Fanuc TP program (LS listing): OP5_LRG_MASTER_AIR_F.LS

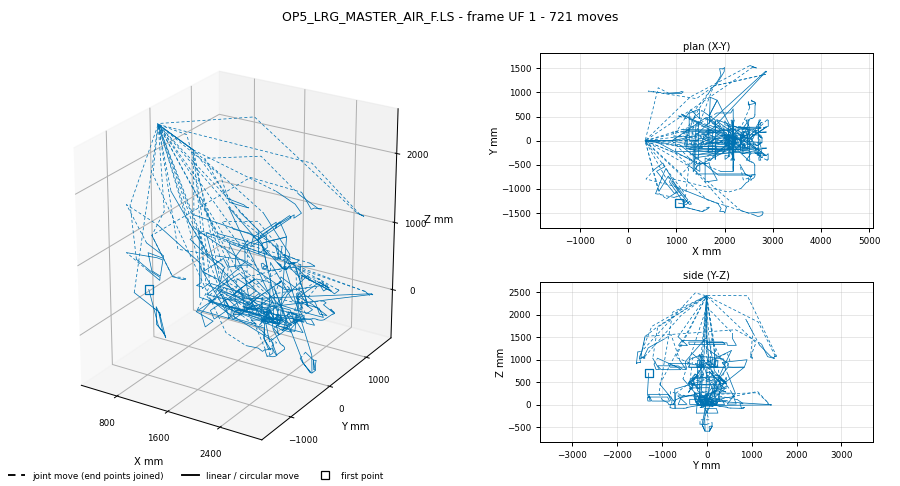
[picture p0: tool path of OP5_LRG_MASTER_AIR_F.LS in frame UF 1, 721 of 721 moves have a stored position in this frame; points joined in program order, loops and branches not executed]
/PROG  OP5_LRG_MASTER_AIR_F
/ATTR
OWNER		= MNEDITOR;
COMMENT		= "Air move update";
PROG_SIZE	= 123886;
CREATE		= DATE 25-08-25  TIME 10:39:22;
MODIFIED	= DATE 25-08-25  TIME 10:43:36;
FILE_NAME	= OP5_LRG_;
VERSION		= 0;
LINE_COUNT	= 2640;
MEMORY_SIZE	= 124514;
PROTECT		= READ_WRITE;
TCD:  STACK_SIZE	= 0,
      TASK_PRIORITY	= 50,
      TIME_SLICE	= 0,
      BUSY_LAMP_OFF	= 0,
      ABORT_REQUEST	= 0,
      PAUSE_REQUEST	= 0;
DEFAULT_GROUP	= 1,1,*,*,*;
CONTROL_CODE	= 00000000 00000000;
/APPL
  ARC Welding Equipment : 1,*,*,*,*;

MPAS ;
MPAS_NUM_PASSES        : 0;
MPAS_LAST_PASS         : 0;
MPAS_CURRENT_PASS      : 0;
MPAS_STATUS_PASS       : 0;
/MN
   1:  !********** WAR HAMMER ********** ;
   2:  !*------- FRAME LARGE ----------* ;
   3:  !*------- FR500 CELL: F --------* ;
   4:  !******************************** ;
   5:   ;
   6:  CALL HOME    ;
   7:  UFRAME_NUM=1 ;
   8:  DO[17:ON :SCAN ZONE2]=OFF ;
   9:   ;
  10:  !********POSITIONER MOVE******** ;
  11:J P[1] 85% CNT30    ;
  12:   ;
  13:L P[3] 1000mm/sec CNT40    ;
  14:   ;
  15:  !FR50L1000 ;
  16:  IF R[15:TECH HOLD]=1002,CALL TECH_HOLD ;
  17:   ;
  18:  !TO SKIP FRONT BUMPER WELDS ;
  19:  CALL ARC_DISABLE_FRONT_BMPR_LRG(0) ;
  20:   ;
1578:   ;
1579:L P[124] 1000mm/sec FINE
    :  Arc Start[6]    ;
1580:  Weave Sine[6] ;
1581:  Track TAST[6] ;
1582:L P[125] WELD_SPEED FINE
    :  Arc End[6]    ;
1583:  Weave End ;
1584:  Track End ;
1585:   ;
  22:   ;
  23:   ;
  24:L P[8] 800mm/sec CNT30    ;
  25:   ;
  26:L P[9] 1000mm/sec CNT30    ;
  27:   ;
  28:   ;
  29:  !FR50L1001 ;
  30:  IF R[15:TECH HOLD]=1003,CALL TECH_HOLD ;
  31:   ;
  32:   ;
1587:   ;
1588:L P[126] 1000mm/sec FINE
    :  Arc Start[6]    ;
1589:  Weave Sine[6] ;
1590:  Track TAST[6] ;
1591:L P[129] WELD_SPEED FINE
    :  Arc End[6]    ;
1592:  Weave End ;
1593:  Track End ;
1594:   ;
  34:   ;
  35:L P[12] 1000mm/sec CNT100    ;
  36:   ;
  37:   ;
  38:  !FR50L1002 ;
  39:  IF R[15:TECH HOLD]=1004,CALL TECH_HOLD ;
  40:   ;
  41:   ;
  42:L P[13] 1000mm/sec CNT70    ;
  43:   ;
1596:   ;
1597:L P[130] 1000mm/sec FINE
    :  Arc Start[6]    ;
1598:  Weave Sine[6] ;
1599:  Track TAST[6] ;
1600:L P[131] WELD_SPEED FINE
    :  Arc End[6]    ;
1601:  Weave End ;
1602:  Track End ;
1603:   ;
  45:   ;
  46:  CALL ARC_DISABLE_FRONT_BMPR_LRG(1) ;
  47:   ;
  48:L P[16] 1000mm/sec CNT100    ;
  49:   ;
  50:  !HOME ;
  51:J P[4] 70% CNT30    ;
  52:   ;
  53:  !********POSITIONER MOVE******** ;
  54:J P[17] 85% CNT30    ;
  55:   ;
  56:J P[18] 50% CNT100    ;
  57:   ;
  58:L P[19] 1000mm/sec CNT100    ;
  59:   ;
  60:   ;
  61:  !FR50L1003 ;
  62:  IF R[15:TECH HOLD]=1005,CALL TECH_HOLD ;
  63:   ;
  64:   ;
  65:L P[20] 1000mm/sec CNT25    ;
  66:   ;
1605:   ;
1606:L P[132] 1000mm/sec FINE
    :  Arc Start[6]    ;
1607:  Weave Sine[6] ;
1608:  Track TAST[6] ;
1609:L P[137] WELD_SPEED CNT100    ;
1610:L P[138] WELD_SPEED FINE
    :  Arc End[6]    ;
1611:  Track End ;
1612:  Weave End ;
1613:   ;
  68:   ;
  69:L P[24] 1000mm/sec CNT30    ;
  70:   ;
  71:   ;
  72:  !FR50L1010 ;
  73:  IF R[15:TECH HOLD]=1012,CALL TECH_HOLD ;
  74:   ;
  75:   ;
  76:L P[25] 1000mm/sec CNT30    ;
  77:   ;
1615:   ;
1616:L P[141] 1000mm/sec FINE
    :  Arc Start[6]    ;
1617:  Weave Sine[6] ;
1618:  Track TAST[6] ;
1619:L P[142] WELD_SPEED CNT100    ;
1620:L P[146] WELD_SPEED FINE
    :  Arc End[6]    ;
1621:  Weave End ;
1622:  Track End ;
1623:   ;
  79:   ;
  80:L P[29] 1000mm/sec CNT25    ;
  81:   ;
  82:   ;
  83:  !FR50L1020 ;
  84:  IF R[15:TECH HOLD]=1022,CALL TECH_HOLD ;
  85:   ;
  86:   ;
  87:J P[30] 50% CNT25    ;
  88:   ;
1625:   ;
1626:L P[147] 1000mm/sec FINE
    :  Arc Start[6]    ;
1627:  Weave Sine[6] ;
1628:  Track TAST[6] ;
1629:L P[150] WELD_SPEED FINE
    :  Arc End[6]    ;
1630:  Weave End ;
1631:  Track End ;
1632:   ;
  90:   ;
  91:L P[33] 1000mm/sec CNT30    ;
  92:   ;
  93:L P[34] 1000mm/sec CNT30    ;
  94:   ;
  95:   ;
  96:  !FR50L1030 ;
  97:  IF R[15:TECH HOLD]=1032,CALL TECH_HOLD ;
  98:   ;
  99:   ;
1634:   ;
1635:L P[151] 1000mm/sec FINE
    :  Arc Start[6]    ;
1636:  Weave Sine[6] ;
1637:  Track TAST[6] ;
1638:L P[156] WELD_SPEED FINE
    :  Arc End[6]    ;
1639:  Weave End ;
1640:  Track End ;
1641:   ;
 101:   ;
 102:L P[37] 1000mm/sec CNT50    ;
 103:   ;
 104:J P[38] 50% CNT50    ;
 105:   ;
 106:L P[39] 1000mm/sec CNT25    ;
 107:   ;
 108:   ;
 109:  !FR50L1040 ;
 110:  IF R[15:TECH HOLD]=1042,CALL TECH_HOLD ;
 111:   ;
 112:   ;
1643:   ;
1644:L P[157] 1000mm/sec FINE
    :  Arc Start[6]    ;
1645:  Weave Sine[6] ;
1646:L P[158] WELD_SPEED FINE
    :  Arc End[6]    ;
1647:  Weave End ;
1648:   ;
 114:   ;
 115:L P[42] 1000mm/sec CNT30    ;
 116:   ;
 117:L P[43] 1000mm/sec CNT70    ;
 118:   ;
 119:J P[44] 50% CNT50    ;
 120:   ;
 121:L P[45] 1000mm/sec CNT30    ;
 122:   ;
 123:   ;
 124:  !FR50L1050 ;
 125:  IF R[15:TECH HOLD]=1052,CALL TECH_HOLD ;
 126:   ;
 127:   ;
1650:   ;
1651:L P[161] 1000mm/sec FINE
    :  Arc Start[6]    ;
1652:  Weave Sine[6] ;
1653:L P[162] WELD_SPEED FINE
    :  Arc End[6]    ;
1654:  Weave End ;
1655:   ;
 129:   ;
 130:L P[48] 1000mm/sec CNT80    ;
 131:   ;
 132:J P[49] 50% CNT25    ;
 133:   ;
 134:L P[50] 1000mm/sec CNT25    ;
 135:   ;
 136:   ;
 137:  !FR50L1060 ;
 138:  IF R[15:TECH HOLD]=1062,CALL TECH_HOLD ;
 139:   ;
 140:   ;
1657:   ;
1658:L P[770] 1000mm/sec FINE
    :  Arc Start[6]    ;
1659:  Weave Sine[6] ;
1660:L P[771] WELD_SPEED FINE
    :  Arc End[6]    ;
1661:  Weave End ;
1662:   ;
 142:   ;
 143:L P[53] 500mm/sec CNT100    ;
 144:   ;
 145:L P[54] 1500mm/sec CNT35    ;
 146:   ;
 147:J P[55] 50% CNT30    ;
 148:   ;
 149:L P[56] 1000mm/sec CNT30    ;
 150:   ;
 151:   ;
 152:  !FR50L1070 ;
 153:  IF R[15:TECH HOLD]=1072,CALL TECH_HOLD ;
 154:   ;
 155:   ;
1664:   ;
1665:L P[772] 1000mm/sec FINE
    :  Arc Start[6]    ;
1666:  Weave Sine[6] ;
1667:  Track TAST[6] ;
1668:L P[773] WELD_SPEED FINE
    :  Arc End[6]    ;
1669:  Weave End ;
1670:  Track End ;
1671:   ;
 157:   ;
 158:L P[59] 1000mm/sec CNT100    ;
 159:   ;
 160:L P[60] 1000mm/sec CNT80    ;
 161:   ;
 162:   ;
 163:  !FR50L1080 ;
 164:  IF R[15:TECH HOLD]=1082,CALL TECH_HOLD ;
 165:   ;
 166:   ;
1673:   ;
1674:L P[774] 1000mm/sec FINE
    :  Arc Start[6]    ;
1675:  Weave Sine[6] ;
1676:  Track TAST[6] ;
1677:L P[775] WELD_SPEED FINE
    :  Arc End[6]    ;
1678:  Weave End ;
1679:  Track End ;
1680:   ;
 168:   ;
 169:J P[63] 30% CNT100    ;
 170:   ;
 171:J P[64] 50% CNT100    ;
 172:   ;
 173:L P[65] 1000mm/sec CNT80    ;
 174:   ;
 175:   ;
 176:  !FR50L1090 ;
 177:  IF R[15:TECH HOLD]=1092,CALL TECH_HOLD ;
 178:  !10MM PASS ;
 179:   ;
 180:   ;
1682:   ;
1683:L P[776] 1000mm/sec FINE
    :  Arc Start[6]    ;
1684:  Weave Sine[6] ;
1685:  Track TAST[6] RPM[1] ;
1686:L P[777] WELD_SPEED CNT100    ;
1687:L P[779] WELD_SPEED CNT100    ;
1688:C P[782]
    :  P[783] WELD_SPEED CNT100    ;
1689:L P[784] WELD_SPEED FINE
    :  Arc End[6]    ;
1690:  Track End ;
1691:  Weave End ;
1692:   ;
 182:   ;
 183:J P[72] 16% CNT25    ;
 184:   ;
 185:J P[74] 50% CNT25    ;
 186:   ;
 187:L P[75] 1000mm/sec CNT25    ;
 188:   ;
 189:   ;
 190:  !FR50L1100 ;
 191:  IF R[15:TECH HOLD]=1102,CALL TECH_HOLD ;
 192:   ;
 193:   ;
1694:   ;
1695:L P[785] 1000mm/sec FINE
    :  Arc Start[6]    ;
1696:  Weave Sine[6] ;
1697:  Track TAST[6] RPM[2] ;
1698:L P[786] WELD_SPEED CNT100    ;
1699:L P[787] WELD_SPEED CNT100    ;
1700:C P[788]
    :  P[789] WELD_SPEED CNT100    ;
1701:L P[791] WELD_SPEED FINE
    :  Arc End[6]    ;
1702:  Weave End ;
1703:  Track End ;
1704:   ;
 195:   ;
 196:J P[82] 30% CNT10    ;
 197:   ;
 198:J P[83] 50% CNT80    ;
 199:   ;
 200:L P[84] 1000mm/sec CNT25    ;
 201:   ;
 202:   ;
 203:  !FR50L1110MP ;
 204:  IF R[15:TECH HOLD]=1112,CALL TECH_HOLD ;
 205:   ;
 206:   ;
 207:  MP Offset  PR[3] RPM[1] ;
 210:   ;
 211:J P[91] 25% CNT10    ;
 212:   ;
 213:J P[92] 50% CNT30    ;
 214:   ;
 215:L P[93] 1000mm/sec CNT25    ;
 216:   ;
 217:   ;
 218:  !FR50M1110MP ;
 219:   ;
 220:   ;
 221:  MP Offset  PR[4] RPM[1] ;
 224:   ;
 225:J P[100] 25% CNT25    ;
 226:   ;
 227:J P[102] 50% CNT25    ;
 228:   ;
 229:L P[103] 1000mm/sec CNT25    ;
 230:   ;
 231:   ;
 232:  !FR50L1120MP ;
 233:  IF R[15:TECH HOLD]=1122,CALL TECH_HOLD ;
 234:   ;
 235:   ;
 236:  MP Offset  PR[1] RPM[2] ;
 239:   ;
 240:J P[110] 50% CNT25    ;
 241:   ;
 242:J P[111] 50% CNT25    ;
 243:   ;
 244:L P[112] 1000mm/sec CNT25    ;
 245:   ;
 246:   ;
 247:  !FR501130MP ;
 248:   ;
 249:   ;
 250:  MP Offset  PR[2] RPM[2] ;
 253:   ;
 254:J P[119] 50% CNT25    ;
 255:   ;
 256:J P[121] 50% CNT25    ;
 257:   ;
 258:L P[122] 1000mm/sec CNT25    ;
 259:   ;
 260:   ;
 261:  !FR50L1140 ;
 262:  IF R[15:TECH HOLD]=1142,CALL TECH_HOLD ;
 263:   ;
 264:   ;
1746:   ;
1747:L P[817] 1000mm/sec FINE
    :  Arc Start[8]    ;
1748:  Weave Sine[8] ;
1749:L P[818] WELD_SPEED CNT100    ;
1750:C P[819]
    :  P[820] WELD_SPEED FINE
    :  Arc End[8]    ;
1751:  Weave End ;
1752:   ;
 266:   ;
 267:L P[127] 1000mm/sec CNT25    ;
 268:   ;
 269:J P[128] 50% CNT25    ;
 270:   ;
 271:   ;
 272:  !FR50L1141 ;
 273:  IF R[15:TECH HOLD]=1143,CALL TECH_HOLD ;
 274:   ;
 275:   ;
1754:   ;
1755:L P[821] 1000mm/sec FINE
    :  Arc Start[8]    ;
1756:  Weave Sine[8] ;
1757:L P[822] WELD_SPEED CNT100    ;
1758:C P[823]
    :  P[824] WELD_SPEED FINE
    :  Arc End[8]    ;
1759:  Weave End ;
1760:   ;
 277:   ;
 278:L P[133] 1000mm/sec CNT25    ;
 279:   ;
 280:L P[134] 1000mm/sec CNT25    ;
 281:   ;
 282:J P[135] 50% CNT25    ;
 283:   ;
 284:L P[136] 1000mm/sec CNT50    ;
 285:   ;
 286:   ;
 287:  !FR50L1150 ;
 288:  IF R[15:TECH HOLD]=1152,CALL TECH_HOLD ;
 289:   ;
 290:   ;
1762:   ;
1763:L P[825] 1000mm/sec FINE
    :  Arc Start[6]    ;
1764:  Weave Sine[6] ;
1765:  Track TAST[6] ;
1766:L P[826] WELD_SPEED FINE
    :  Arc End[6]    ;
1767:  Weave End ;
1768:  Track End ;
1769:   ;
 292:   ;
 293:L P[139] 1000mm/sec CNT100    ;
 294:   ;
 295:L P[140] 1000mm/sec CNT50    ;
 296:   ;
 297:   ;
 298:  !FR50L1160 ;
 299:  IF R[15:TECH HOLD]=1162,CALL TECH_HOLD ;
 300:   ;
1771:   ;
1772:L P[827] 1000mm/sec FINE
    :  Arc Start[6]    ;
1773:  Weave Sine[6] ;
1774:  Track TAST[6] ;
1775:L P[828] WELD_SPEED FINE
    :  Arc End[6]    ;
1776:  Weave End ;
1777:  Track End ;
1778:   ;
 302:   ;
 303:L P[143] 1000mm/sec CNT30    ;
 304:   ;
 305:  !********POSITIONER MOVE******** ;
 306:J P[144] 85% CNT30    ;
 307:   ;
 308:L P[145] 1000mm/sec CNT100    ;
 309:   ;
 310:   ;
 311:  !FR50L1170 ;
 312:  IF R[15:TECH HOLD]=1172,CALL TECH_HOLD ;
 313:   ;
 314:   ;
1780:   ;
1781:L P[829] 1000mm/sec FINE
    :  Arc Start[6]    ;
1782:  Weave Sine[6] ;
1783:  Track TAST[6] ;
1784:L P[830] WELD_SPEED FINE
    :  Arc End[6]    ;
1785:  Weave End ;
1786:  Track End ;
1787:   ;
 316:   ;
 317:L P[148] 1000mm/sec CNT100    ;
 318:   ;
 319:L P[149] 1500mm/sec CNT100    ;
 320:   ;
 321:   ;
 322:  !FR50L1180 ;
 323:  IF R[15:TECH HOLD]=1182,CALL TECH_HOLD ;
 324:   ;
 325:   ;
1789:   ;
1790:L P[831] 1000mm/sec FINE
    :  Arc Start[6]    ;
1791:  Weave Sine[6] ;
1792:  Track TAST[6] ;
1793:L P[832] WELD_SPEED FINE
    :  Arc End[6]    ;
1794:  Weave End ;
1795:  Track End ;
1796:   ;
 327:   ;
 328:L P[152] 1000mm/sec CNT100    ;
 329:   ;
 330:  !HOME ;
 331:J P[7] 100% CNT30    ;
 332:  TIMER[7]=RESET ;
 333:  TIMER[7]=START ;
 334:   ;
 335:  !********POSITIONER MOVE******** ;
 336:J P[153] 80% CNT30    ;
 337:   ;
 338:J P[154] 50% CNT100    ;
 339:   ;
 340:L P[155] 1000mm/sec CNT25    ;
 341:   ;
 342:   ;
 343:  !FR50L1210 ;
 344:  IF R[15:TECH HOLD]=1212,CALL TECH_HOLD ;
 345:   ;
 346:   ;
1798:   ;
1799:L P[833] 1000mm/sec FINE
    :  Arc Start[6]    ;
1800:  Weave Sine[6] ;
1801:  Track TAST[6] ;
1802:L P[834] WELD_SPEED CNT100    ;
1803:L P[835] WELD_SPEED FINE
    :  Arc End[6]    ;
1804:  Weave End ;
1805:  Track End ;
1806:   ;
 348:   ;
 349:L P[159] 1000mm/sec CNT25    ;
 350:   ;
 351:L P[160] 1000mm/sec CNT25    ;
 352:   ;
 353:   ;
 354:  !FR50L1220 ;
 355:  IF R[15:TECH HOLD]=1222,CALL TECH_HOLD ;
 356:   ;
 357:   ;
1808:   ;
1809:L P[836] 1000mm/sec FINE
    :  Arc Start[6]    ;
1810:  Weave Sine[6] ;
1811:  Track TAST[6] ;
1812:L P[837] WELD_SPEED CNT100    ;
1813:L P[838] WELD_SPEED FINE
    :  Arc End[6]    ;
1814:  Weave End ;
1815:  Track End ;
1816:   ;
 359:   ;
 360:L P[163] 1000mm/sec CNT80    ;
 361:   ;
 362:L P[164] 1200mm/sec CNT25    ;
 363:   ;
 364:   ;
 365:  !FR50L1230 ;
 366:  IF R[15:TECH HOLD]=1232,CALL TECH_HOLD ;
 367:   ;
 368:   ;
1818:   ;
1819:L P[839] 1000mm/sec FINE
    :  Arc Start[6]    ;
1820:  Weave Sine[6] ;
1821:  Track TAST[6] ;
1822:L P[840] WELD_SPEED CNT100    ;
1823:L P[841] WELD_SPEED FINE
    :  Arc End[6]    ;
1824:  Weave End ;
1825:  Track End ;
1826:   ;
 370:   ;
 371:L P[167] 1000mm/sec CNT25    ;
 372:   ;
 373:L P[168] 1000mm/sec CNT25    ;
 374:   ;
 375:   ;
 376:  !FR50L1240 ;
 377:  IF R[15:TECH HOLD]=1242,CALL TECH_HOLD ;
 378:   ;
 379:   ;
1828:   ;
1829:L P[842] 1000mm/sec FINE
    :  Arc Start[6]    ;
1830:  Weave Sine[6] ;
1831:  Track TAST[6] ;
1832:L P[843] WELD_SPEED CNT100    ;
1833:L P[844] WELD_SPEED FINE
    :  Arc End[6]    ;
1834:  Weave End ;
1835:  Track End ;
1836:   ;
 381:   ;
 382:L P[172] 1000mm/sec CNT25    ;
 383:   ;
 384:L P[173] 1000mm/sec CNT100    ;
 385:   ;
 386:  !HOME ;
 387:J P[116] 100% CNT100    ;
 388:   ;
 389:   ;
 390:  !********POSITIONER MOVE******** ;
 391:J P[174] 85% FINE    ;
 392:   ;
 393:  CALL T_CLEAN    ;
 394:   ;
 395:J P[175] 50% CNT35    ;
 396:   ;
 397:L P[176] 1000mm/sec CNT25    ;
 398:   ;
 399:   ;
 400:  !FR50L1250 ;
 401:  IF R[15:TECH HOLD]=1252,CALL TECH_HOLD ;
 402:   ;
 403:   ;
1838:   ;
1839:L P[845] 1000mm/sec FINE
    :  Arc Start[6]    ;
1840:  Weave Sine[6] ;
1841:  Track TAST[6] ;
1842:L P[846] WELD_SPEED CNT100    ;
1843:L P[847] WELD_SPEED CNT100    ;
1844:L P[848] WELD_SPEED FINE
    :  Arc End[6]    ;
1845:  Weave End ;
1846:  Track End ;
1847:   ;
 405:   ;
 406:L P[181] 1000mm/sec CNT100    ;
 407:   ;
 408:J P[182] 50% CNT100    ;
 409:   ;
 410:L P[184] 500mm/sec CNT100    ;
 411:   ;
 412:   ;
 413:  !FR50L1260 ;
 414:  IF R[15:TECH HOLD]=1262,CALL TECH_HOLD ;
 415:   ;
 416:   ;
1849:   ;
1850:L P[849] 1000mm/sec FINE
    :  Arc Start[6]    ;
1851:  Weave Sine[6] ;
1852:  Track TAST[6] ;
1853:L P[850] WELD_SPEED CNT100    ;
1854:L P[851] WELD_SPEED CNT100    ;
1855:L P[852] WELD_SPEED FINE
    :  Arc End[6]    ;
1856:  Weave End ;
1857:  Track End ;
1858:   ;
 418:   ;
 419:L P[189] 1000mm/sec CNT25    ;
 420:   ;
 421:J P[190] 50% CNT25    ;
 422:   ;
 423:L P[191] 1000mm/sec CNT25    ;
 424:   ;
 425:   ;
 426:  !FR50L1270 ;
 427:  IF R[15:TECH HOLD]=1272,CALL TECH_HOLD ;
 428:   ;
 429:   ;
1860:   ;
1861:L P[853] 1000mm/sec FINE
    :  Arc Start[6]    ;
1862:  Weave Sine[6] ;
1863:  Track TAST[6] ;
1864:L P[854] WELD_SPEED CNT100    ;
1865:  Track End ;
1866:L P[855] WELD_SPEED FINE
    :  Arc End[6]    ;
1867:  Weave End ;
1868:  Track End ;
1869:   ;
 431:   ;
 432:L P[195] 1000mm/sec CNT80    ;
 433:   ;
 434:L P[196] 1000mm/sec CNT100    ;
 435:   ;
 436:   ;
 437:  !FR50L1280 ;
 438:  IF R[15:TECH HOLD]=1282,CALL TECH_HOLD ;
 439:   ;
 440:   ;
1871:   ;
1872:L P[856] 1000mm/sec FINE
    :  Arc Start[6]    ;
1873:  Weave Sine[6] ;
1874:  Track TAST[6] ;
1875:L P[857] WELD_SPEED CNT100    ;
1876:  Track End ;
1877:L P[858] WELD_SPEED FINE
    :  Arc End[6]    ;
1878:  Weave End ;
1879:  Track End ;
1880:   ;
 442:   ;
 443:L P[200] 1000mm/sec CNT25    ;
 444:   ;
 445:J P[201] 50% CNT25    ;
 446:   ;
 447:L P[202] 1000mm/sec CNT25    ;
 448:  TIMER[7]=RESET ;
 449:  TIMER[7]=START ;
 450:   ;
 451:   ;
 452:  !FR50L1290 ;
 453:  IF R[15:TECH HOLD]=1292,CALL TECH_HOLD ;
 454:   ;
 455:   ;
1882:   ;
1883:L P[859] 1000mm/sec FINE
    :  Arc Start[6]    ;
1884:  Weave Sine[6] ;
1885:  Track TAST[6] ;
1886:L P[860] WELD_SPEED CNT100    ;
1887:L P[861] WELD_SPEED FINE
    :  Arc End[6]    ;
1888:  Weave End ;
1889:  Track End ;
1890:   ;
 457:   ;
 458:L P[206] 1000mm/sec CNT100    ;
 459:   ;
 460:L P[207] 1000mm/sec CNT100    ;
 461:   ;
 462:   ;
 463:  !FR50L1300 ;
 464:  IF R[15:TECH HOLD]=1302,CALL TECH_HOLD ;
 465:   ;
 466:   ;
1892:   ;
1893:L P[862] 1000mm/sec FINE
    :  Arc Start[6]    ;
1894:  Weave Sine[6] ;
1895:  Track TAST[6] ;
1896:L P[863] WELD_SPEED CNT100    ;
1897:L P[864] WELD_SPEED FINE
    :  Arc End[6]    ;
1898:  Weave End ;
1899:  Track End ;
1900:   ;
 468:   ;
 469:L P[210] 1000mm/sec CNT100    ;
 470:   ;
 471:L P[211] 1000mm/sec CNT100    ;
 472:   ;
 473:   ;
 474:  !FR50L1310 ;
 475:  IF R[15:TECH HOLD]=1312,CALL TECH_HOLD ;
 476:   ;
 477:   ;
1902:   ;
1903:L P[865] 1000mm/sec FINE
    :  Arc Start[6]    ;
1904:  Weave Sine[6] ;
1905:  Track TAST[6] ;
1906:L P[866] WELD_SPEED FINE
    :  Arc End[6]    ;
1907:  Weave End ;
1908:  Track End ;
1909:   ;
 479:   ;
 480:L P[214] 1000mm/sec CNT100    ;
 481:   ;
 482:L P[215] 1000mm/sec CNT100    ;
 483:   ;
 484:   ;
 485:  !FR50L1320 ;
 486:  IF R[15:TECH HOLD]=1322,CALL TECH_HOLD ;
 487:   ;
 488:   ;
1911:   ;
1912:L P[867] 1000mm/sec FINE
    :  Arc Start[6]    ;
1913:  Weave Sine[6] ;
1914:  Track TAST[6] ;
1915:L P[868] WELD_SPEED CNT100    ;
1916:L P[869] WELD_SPEED FINE
    :  Arc End[6]    ;
1917:  Weave End ;
1918:  Track End ;
1919:   ;
 490:   ;
 491:L P[219] 1000mm/sec CNT100    ;
 492:   ;
 493:L P[220] 1000mm/sec CNT100    ;
 494:  TIMER[7]=STOP ;
 495:   ;
 496:J P[73] 50% CNT30    ;
 497:   ;
 498:  !********POSITIONER MOVE******** ;
 499:J P[86] 100% CNT30    ;
 500:   ;
 501:  !FR50L1330 ;
 502:  IF R[15:TECH HOLD]=1332,CALL TECH_HOLD ;
 503:   ;
 504:   ;
 505:J P[327] 40% CNT10    ;
 506:   ;
1921:   ;
1922:L P[870] 1000mm/sec FINE
    :  Arc Start[8]    ;
1923:  Weave Sine[8] ;
1924:L P[871] WELD_SPEED FINE
    :  Arc End[8]    ;
1925:  Weave End ;
1926:   ;
 508:   ;
 509:J P[85] 50% CNT30    ;
 510:   ;
 511:J P[87] 50% CNT20    ;
 512:   ;
 513:  !********POSITIONER MOVE******** ;
 514:J P[225] 80% CNT20    ;
 515:   ;
 516:   ;
 517:   ;
 518:  !FR50L1340 ;
 519:  IF R[15:TECH HOLD]=1342,CALL TECH_HOLD ;
 520:   ;
 521:   ;
1928:   ;
1929:L P[872] 1000mm/sec FINE
    :  Arc Start[6]    ;
1930:  Weave Sine[6] ;
1931:L P[873] WELD_SPEED FINE
    :  Arc End[6]    ;
1932:  Weave End ;
1933:   ;
 523:   ;
 524:   ;
 525:  !FR50L1350 ;
 526:  IF R[15:TECH HOLD]=1352,CALL TECH_HOLD ;
 527:   ;
 528:   ;
1935:   ;
1936:L P[874] 1000mm/sec FINE
    :  Arc Start[6]    ;
1937:  Weave Sine[6] ;
1938:L P[875] WELD_SPEED FINE
    :  Arc End[6]    ;
1939:  Weave End ;
1940:   ;
 530:   ;
 531:L P[230] 1000mm/sec CNT25    ;
 532:   ;
 533:  !HOME ;
 534:J P[117] 100% CNT50    ;
 535:   ;
 536:  !********POSITIONER MOVE******** ;
 537:J P[231] 90% CNT25    ;
 538:   ;
 539:J P[232] 50% CNT25    ;
 540:   ;
 541:L P[234] 1000mm/sec CNT25    ;
 542:   ;
 543:J P[235] 50% CNT25    ;
 544:   ;
 545:   ;
 546:  !FR50L1380 ;
 547:  IF R[15:TECH HOLD]=1382,CALL TECH_HOLD ;
 548:   ;
 549:   ;
1942:   ;
1943:L P[876] 1000mm/sec FINE
    :  Arc Start[6]    ;
1944:  Weave Sine[6] ;
1945:  Track TAST[6] ;
1946:L P[877] WELD_SPEED CNT100    ;
1947:L P[878] WELD_SPEED CNT100    ;
1948:L P[879] WELD_SPEED FINE
    :  Arc End[6]    ;
1949:  Weave End ;
1950:  Track End ;
1951:   ;
 551:   ;
 552:L P[240] 800mm/sec CNT2    ;
 553:   ;
 554:L P[241] 800mm/sec CNT25    ;
 555:   ;
 556:  !********POSITIONER MOVE******** ;
 557:J P[242] 75% CNT5    ;
 558:   ;
 559:L P[243] 1000mm/sec CNT25    ;
 560:   ;
 561:   ;
 562:  !FR50L1390 ;
 563:  IF R[15:TECH HOLD]=1392,CALL TECH_HOLD ;
 564:   ;
1953:   ;
1954:L P[880] 1000mm/sec FINE
    :  Arc Start[6]    ;
1955:  Weave Sine[6] ;
1956:L P[881] WELD_SPEED CNT100    ;
1957:L P[882] WELD_SPEED CNT100    ;
1958:L P[883] WELD_SPEED FINE
    :  Arc End[6]    ;
1959:  Weave End ;
1960:   ;
 566:   ;
 567:L P[248] 1000mm/sec CNT25    ;
 568:   ;
 569:L P[249] 1000mm/sec CNT25    ;
 570:   ;
 571:   ;
 572:  !FR50L1400 ;
 573:  IF R[15:TECH HOLD]=1402,CALL TECH_HOLD ;
 574:   ;
 575:   ;
1962:   ;
1963:L P[884] 1000mm/sec FINE
    :  Arc Start[6]    ;
1964:  Weave Sine[6] ;
1965:  Track TAST[6] ;
1966:L P[885] WELD_SPEED FINE
    :  Arc End[6]    ;
1967:  Weave End ;
1968:  Track End ;
1969:   ;
 577:   ;
 578:L P[252] 1000mm/sec CNT25    ;
 579:   ;
 580:   ;
 581:  !FR50L1410 ;
 582:  IF R[15:TECH HOLD]=1412,CALL TECH_HOLD ;
 583:   ;
 584:   ;
1971:   ;
1972:L P[886] 1000mm/sec FINE
    :  Arc Start[6]    ;
1973:  Weave Sine[6] ;
1974:  Track TAST[6] ;
1975:L P[887] WELD_SPEED CNT100    ;
1976:L P[888] WELD_SPEED FINE
    :  Arc End[6]    ;
1977:  Weave End ;
1978:  Track End ;
1979:   ;
 586:   ;
 587:L P[256] 1000mm/sec CNT25    ;
 588:   ;
 589:   ;
 590:  !FR50L1420 ;
 591:  IF R[15:TECH HOLD]=1422,CALL TECH_HOLD ;
 592:   ;
 593:   ;
1981:   ;
1982:L P[889] 1000mm/sec FINE
    :  Arc Start[6]    ;
1983:  Weave Sine[6] ;
1984:  Track TAST[6] ;
1985:L P[890] WELD_SPEED CNT100    ;
1986:L P[891] WELD_SPEED FINE
    :  Arc End[6]    ;
1987:  Weave End ;
1988:  Track End ;
1989:   ;
 595:   ;
 596:L P[260] 1000mm/sec CNT25    ;
 597:   ;
 598:L P[261] 1000mm/sec CNT25    ;
 599:   ;
 600:   ;
 601:  !FR50L1430 ;
 602:  IF R[15:TECH HOLD]=1432,CALL TECH_HOLD ;
 603:   ;
 604:   ;
1991:   ;
1992:L P[892] 1000mm/sec FINE
    :  Arc Start[6]    ;
1993:  Weave Sine[6] ;
1994:L P[893] WELD_SPEED CNT100    ;
1995:  Weave End ;
1996:L P[894] WELD_SPEED FINE
    :  Arc End[6]    ;
1997:   ;
 606:   ;
 607:L P[265] 1000mm/sec CNT25    ;
 608:   ;
 609:   ;
 610:  !FR50L1431 ;
 611:  IF R[15:TECH HOLD]=1433,CALL TECH_HOLD ;
 612:   ;
 613:   ;
1999:   ;
2000:L P[895] 1000mm/sec FINE
    :  Arc Start[6]    ;
2001:  Weave Sine[6] ;
2002:L P[896] WELD_SPEED CNT100    ;
2003:L P[897] WELD_SPEED FINE
    :  Arc End[6]    ;
2004:  Weave End ;
2005:   ;
 615:   ;
 616:L P[269] 1000mm/sec CNT25    ;
 617:   ;
 618:L P[270] 1000mm/sec CNT25    ;
 619:   ;
 620:L P[271] 1000mm/sec CNT50 Wjnt    ;
 621:   ;
 622:J P[272] 50% CNT25    ;
 623:   ;
 624:L P[273] 1000mm/sec CNT25    ;
 625:   ;
 626:   ;
 627:  !FR50L1440 ;
 628:  IF R[15:TECH HOLD]=1442,CALL TECH_HOLD ;
 629:   ;
 630:   ;
2007:   ;
2008:L P[898] 1000mm/sec FINE
    :  Arc Start[6]    ;
2009:  Weave Sine[6] ;
2010:  Track TAST[6] ;
2011:L P[899] WELD_SPEED FINE
    :  Arc End[6]    ;
2012:  Weave End ;
2013:  Track End ;
2014:   ;
 632:   ;
 633:L P[276] 1000mm/sec CNT25    ;
 634:   ;
 635:   ;
 636:  !FR50L1450 ;
 637:  IF R[15:TECH HOLD]=1452,CALL TECH_HOLD ;
 638:   ;
 639:   ;
2016:   ;
2017:L P[900] 1000mm/sec FINE
    :  Arc Start[6]    ;
2018:  Weave Sine[6] ;
2019:  Track TAST[6] ;
2020:L P[901] WELD_SPEED CNT100    ;
2021:L P[902] WELD_SPEED FINE
    :  Arc End[6]    ;
2022:  Weave End ;
2023:  Track End ;
2024:   ;
 641:   ;
 642:L P[280] 1000mm/sec CNT25    ;
 643:   ;
 644:L P[281] 1000mm/sec CNT25    ;
 645:   ;
 646:   ;
 647:  !FR50L1460 ;
 648:  IF R[15:TECH HOLD]=1462,CALL TECH_HOLD ;
 649:   ;
 650:   ;
2026:   ;
2027:L P[903] 1000mm/sec FINE
    :  Arc Start[6]    ;
2028:  Weave Sine[6] ;
2029:  Track TAST[6] ;
2030:L P[904] WELD_SPEED CNT100    ;
2031:L P[905] WELD_SPEED FINE
    :  Arc End[6]    ;
2032:  Weave End ;
2033:  Track End ;
2034:   ;
 652:   ;
 653:L P[285] 1000mm/sec CNT25    ;
 654:   ;
 655:  !********POSITIONER MOVE******** ;
 656:J P[286] 75% FINE    ;
 657:   ;
 658:L P[287] 1000mm/sec CNT25    ;
 659:   ;
 660:   ;
 661:  !FR50L1470 ;
 662:  IF R[15:TECH HOLD]=1472,CALL TECH_HOLD ;
 663:   ;
 664:   ;
2036:   ;
2037:L P[906] 1000mm/sec FINE
    :  Arc Start[6]    ;
2038:  Weave Sine[6] ;
2039:  Track TAST[6] ;
2040:L P[907] WELD_SPEED FINE
    :  Arc End[6]    ;
2041:  Weave End ;
2042:  Track End ;
2043:   ;
 666:   ;
 667:L P[290] 1000mm/sec CNT25    ;
 668:   ;
 669:  !********POSITIONER MOVE******** ;
 670:J P[291] 65% CNT2    ;
 671:   ;
 672:L P[292] 1000mm/sec CNT25    ;
 673:   ;
 674:   ;
 675:  !FR50L1480 ;
 676:  IF R[15:TECH HOLD]=1482,CALL TECH_HOLD ;
 677:   ;
 678:   ;
2045:   ;
2046:L P[908] 1000mm/sec FINE
    :  Arc Start[8]    ;
2047:  Weave Sine[8] ;
2048:L P[909] WELD_SPEED FINE
    :  Arc End[8]    ;
2049:  Weave End ;
2050:   ;
 680:   ;
 681:L P[295] 1000mm/sec CNT25    ;
 682:   ;
 683:L P[296] 1000mm/sec CNT25    ;
 684:   ;
 685:   ;
 686:  !FR50L1490 ;
 687:  IF R[15:TECH HOLD]=1492,CALL TECH_HOLD ;
 688:   ;
 689:   ;
2052:   ;
2053:L P[910] 1000mm/sec FINE
    :  Arc Start[6]    ;
2054:  Weave Sine[6] ;
2055:  Track TAST[6] ;
2056:L P[911] WELD_SPEED FINE
    :  Arc End[6]    ;
2057:  Weave End ;
2058:  Track End ;
2059:   ;
 691:   ;
 692:L P[299] 1000mm/sec CNT25    ;
 693:   ;
 694:L P[300] 1000mm/sec CNT25    ;
 695:   ;
 696:L P[301] 1000mm/sec CNT25    ;
 697:   ;
 698:  !********POSITIONER MOVE******** ;
 699:J P[302] 85% FINE    ;
 700:   ;
 701:L P[303] 1000mm/sec CNT25    ;
 702:   ;
 703:   ;
 704:  !FR50L1500 ;
 705:  IF R[15:TECH HOLD]=1502,CALL TECH_HOLD ;
 706:   ;
 707:   ;
2061:   ;
2062:L P[912] 1000mm/sec FINE
    :  Arc Start[6]    ;
2063:  Weave Sine[6] ;
2064:L P[913] WELD_SPEED CNT100    ;
2065:L P[914] WELD_SPEED FINE
    :  Arc End[6]    ;
2066:  Weave End ;
2067:   ;
 709:   ;
 710:L P[307] 1000mm/sec CNT25    ;
 711:   ;
 712:J P[308] 50% CNT25    ;
 713:   ;
 714:L P[309] 1000mm/sec CNT25    ;
 715:   ;
 716:   ;
 717:  !FR50L1510 ;
 718:  IF R[15:TECH HOLD]=1512,CALL TECH_HOLD ;
 719:   ;
 720:   ;
2069:   ;
2070:L P[915] 1000mm/sec FINE
    :  Arc Start[6]    ;
2071:  Weave Sine[6] ;
2072:  Track TAST[6] ;
2073:L P[916] WELD_SPEED CNT100    ;
2074:C P[917]
    :  P[918] WELD_SPEED CNT100    ;
2075:L P[919] WELD_SPEED CNT100    ;
2076:C P[920]
    :  P[921] WELD_SPEED CNT100    ;
2077:L P[922] WELD_SPEED CNT100    ;
2078:C P[923]
    :  P[924] WELD_SPEED CNT100    ;
2079:L P[925] WELD_SPEED FINE
    :  Arc End[6]    ;
2080:  Weave End ;
2081:  Track End ;
2082:L P[926] 2400mm/sec FINE
    :  Arc Start[1]    ;
2083:L P[927] WELD_SPEED FINE
    :  Arc End[1]    ;
2084:J P[928] 40% FINE
    :  Arc Start[1]    ;
2085:L P[929] WELD_SPEED FINE
    :  Arc End[1]    ;
2086:J P[930] 40% FINE
    :  Arc Start[1]    ;
2087:L P[931] WELD_SPEED FINE
    :  Arc End[1]    ;
2088:   ;
 722:   ;
 723:L P[321] 1000mm/sec CNT25    ;
 724:   ;
 725:J P[322] 40% CNT100    ;
 726:   ;
 727:J P[323] 40% CNT25    ;
 728:   ;
 729:  !CELL ID: F -.. ;
 730:   ;
 731:   ;
 732:J P[324] 50% CNT20    ;
 733:   ;
 740:   ;
 741:L P[328] 800mm/sec CNT25    ;
 742:   ;
 743:J P[224] 40% CNT100    ;
 744:   ;
 745:J P[329] 40% CNT100    ;
 746:   ;
 747:J P[331] 50% CNT50    ;
 748:   ;
 749:L P[332] 1000mm/sec CNT25    ;
 750:   ;
 751:   ;
 752:  !FR50L1520 ;
 753:  IF R[15:TECH HOLD]=1522,CALL TECH_HOLD ;
 754:   ;
 755:   ;
2090:   ;
2091:L P[932] 1000mm/sec FINE
    :  Arc Start[6]    ;
2092:  Weave Sine[6] ;
2093:  Track TAST[6] ;
2094:L P[933] WELD_SPEED FINE
    :  Arc End[6]    ;
2095:  Weave End ;
2096:  Track End ;
2097:   ;
 757:   ;
 758:L P[335] 1000mm/sec CNT25    ;
 759:   ;
 760:J P[336] 50% CNT25    ;
 761:   ;
 762:L P[337] 1000mm/sec CNT25    ;
 763:   ;
 764:   ;
 765:  !FR50L1530 ;
 766:  IF R[15:TECH HOLD]=1532,CALL TECH_HOLD ;
 767:   ;
 768:   ;
2099:   ;
2100:L P[934] 1000mm/sec FINE
    :  Arc Start[6]    ;
2101:  Weave Sine[6] ;
2102:  Track TAST[6] ;
2103:L P[935] WELD_SPEED FINE
    :  Arc End[6]    ;
2104:  Weave End ;
2105:  Track End ;
2106:   ;
 770:   ;
 771:L P[340] 1000mm/sec CNT25    ;
 772:   ;
 773:L P[341] 1000mm/sec CNT25    ;
 774:   ;
 775:L P[342] 1000mm/sec CNT25    ;
 776:   ;
 777:  !FR50L1540 ;
 778:  IF R[15:TECH HOLD]=1542,CALL TECH_HOLD ;
 779:   ;
 780:   ;
2118:   ;
2119:L P[939] 1000mm/sec FINE
    :  Arc Start[6]    ;
2120:  Weave Sine[6] ;
2121:  Track TAST[6] ;
2122:L P[940] WELD_SPEED CNT100    ;
2123:L P[941] WELD_SPEED CNT100    ;
2124:L P[942] WELD_SPEED CNT100    ;
2125:L P[943] WELD_SPEED CNT100    ;
2126:L P[944] WELD_SPEED CNT100    ;
2127:L P[945] WELD_SPEED CNT100    ;
2128:L P[946] WELD_SPEED FINE
    :  Arc End[6]    ;
2129:  Weave End ;
2130:  Track End ;
2131:   ;
 782:   ;
 783:L P[346] 1000mm/sec CNT25    ;
 784:   ;
 785:L P[347] 1000mm/sec CNT25    ;
 786:   ;
 787:L P[348] 1000mm/sec CNT100    ;
 788:   ;
 789:  !HOME ;
 790:J P[118] 100% CNT30    ;
 791:   ;
 792:  !********POSITIONER MOVE******** ;
 793:J P[349] 90% CNT30    ;
 794:   ;
 795:J P[350] 50% CNT25    ;
 796:   ;
 797:L P[351] 1000mm/sec CNT25    ;
 798:   ;
 799:   ;
 800:  !FR50L1540 ;
 801:  IF R[15:TECH HOLD]=1542,CALL TECH_HOLD ;
 802:   ;
 803:   ;
2118:   ;
2119:L P[939] 1000mm/sec FINE
    :  Arc Start[6]    ;
2120:  Weave Sine[6] ;
2121:  Track TAST[6] ;
2122:L P[940] WELD_SPEED CNT100    ;
2123:L P[941] WELD_SPEED CNT100    ;
2124:L P[942] WELD_SPEED CNT100    ;
2125:L P[943] WELD_SPEED CNT100    ;
2126:L P[944] WELD_SPEED CNT100    ;
2127:L P[945] WELD_SPEED CNT100    ;
2128:L P[946] WELD_SPEED FINE
    :  Arc End[6]    ;
2129:  Weave End ;
2130:  Track End ;
2131:   ;
 805:   ;
 806:L P[360] 1000mm/sec CNT60    ;
 807:   ;
 808:L P[361] 1000mm/sec CNT25    ;
 809:   ;
 810:   ;
 811:  !FR50L1550 ;
 812:  IF R[15:TECH HOLD]=1552,CALL TECH_HOLD ;
 813:   ;
 814:   ;
2133:   ;
2134:L P[947] 1000mm/sec FINE
    :  Arc Start[6]    ;
2135:  Weave Sine[6] ;
2136:  Track TAST[6] ;
2137:L P[948] WELD_SPEED CNT100    ;
2138:L P[949] WELD_SPEED CNT100    ;
2139:L P[950] WELD_SPEED CNT100    ;
2140:L P[951] WELD_SPEED FINE
    :  Arc End[6]    ;
2141:  Weave End ;
2142:  Track End ;
2143:   ;
 816:   ;
 817:L P[367] 1000mm/sec CNT25    ;
 818:   ;
 819:L P[368] 1000mm/sec CNT100    ;
 820:   ;
 821:  !HOME ;
 822:J P[183] 100% CNT60    ;
 823:   ;
 824:  !********POSITIONER MOVE******** ;
 825:  !LOAD POSITION ;
 826:J P[233] 90% FINE    ;
 827:   ;
 828:  CALL HOME    ;
 829:  CALL T_CLEAN    ;
 830:   ;
 831:  !********POSITIONER MOVE******** ;
 832:J P[377] 90% CNT20    ;
 833:   ;
 834:L P[378] 1000mm/sec CNT25    ;
 835:   ;
 836:L P[379] 1000mm/sec CNT25    ;
 837:   ;
 838:   ;
 839:  !FR50L1570 ;
 840:  IF R[15:TECH HOLD]=1572,CALL TECH_HOLD ;
 841:   ;
 842:   ;
2145:   ;
2146:L P[952] 1000mm/sec FINE
    :  Arc Start[6]    ;
2147:  Weave Sine[6] ;
2148:  Track TAST[6] ;
2149:L P[953] WELD_SPEED CNT100    ;
2150:L P[954] WELD_SPEED CNT100    ;
2151:L P[955] WELD_SPEED CNT100    ;
2152:L P[956] WELD_SPEED CNT100    ;
2153:L P[957] WELD_SPEED CNT100    ;
2154:L P[958] WELD_SPEED CNT100    ;
2155:L P[959] WELD_SPEED FINE
    :  Arc End[6]    ;
2156:  Weave End ;
2157:  Track End ;
2158:   ;
 844:   ;
 845:L P[388] 1000mm/sec CNT100    ;
 846:   ;
 847:L P[389] 1000mm/sec CNT25    ;
 848:   ;
 849:   ;
 850:  !FR50L1580 ;
 851:  IF R[15:TECH HOLD]=1582,CALL TECH_HOLD ;
 852:   ;
 853:   ;
2160:   ;
2161:L P[960] 1000mm/sec FINE
    :  Arc Start[6]    ;
2162:  Weave Sine[6] ;
2163:  Track TAST[6] ;
2164:L P[961] WELD_SPEED CNT100    ;
2165:L P[962] WELD_SPEED CNT100    ;
2166:L P[963] WELD_SPEED CNT100    ;
2167:L P[964] WELD_SPEED FINE
    :  Arc End[6]    ;
2168:  Weave End ;
2169:  Track End ;
2170:   ;
 855:   ;
 856:L P[395] 600mm/sec CNT25    ;
 857:   ;
 858:L P[396] 1000mm/sec CNT100    ;
 859:   ;
 860:J P[326] 100% CNT25    ;
 861:   ;
 862:J P[325] 100% CNT30    ;
 863:   ;
 864:  !********POSITIONER MOVE******** ;
 865:J P[397] 90% CNT30    ;
 866:   ;
 867:J P[398] 50% CNT100    ;
 868:   ;
 869:L P[399] 1000mm/sec CNT25    ;
 870:   ;
 871:   ;
 872:  !FR50L1590 ;
 873:  IF R[15:TECH HOLD]=1592,CALL TECH_HOLD ;
 874:   ;
 875:   ;
2172:   ;
2173:L P[965] 1000mm/sec FINE
    :  Arc Start[6]    ;
2174:  Weave Sine[6] ;
2175:  Track TAST[6] ;
2176:L P[966] WELD_SPEED FINE
    :  Arc End[6]    ;
2177:  Weave End ;
2178:  Track End ;
2179:   ;
 877:   ;
 878:L P[402] 1000mm/sec CNT25    ;
 879:   ;
 880:J P[403] 50% CNT25    ;
 881:   ;
 882:   ;
 883:  !FR50L1600 ;
 884:  IF R[15:TECH HOLD]=1602,CALL TECH_HOLD ;
 885:   ;
 886:   ;
2181:   ;
2182:L P[967] 1000mm/sec FINE
    :  Arc Start[6]    ;
2183:  Weave Sine[6] ;
2184:  Track TAST[6] ;
2185:L P[968] WELD_SPEED FINE
    :  Arc End[6]    ;
2186:  Weave End ;
2187:  Track End ;
2188:   ;
 888:   ;
 889:L P[406] 1000mm/sec CNT25    ;
 890:   ;
 891:J P[407] 50% CNT25    ;
 892:   ;
 893:   ;
 894:  !FR50L1601 ;
 895:  IF R[15:TECH HOLD]=1603,CALL TECH_HOLD ;
 896:   ;
 897:   ;
2190:   ;
2191:L P[969] 1000mm/sec FINE
    :  Arc Start[6]    ;
2192:  Weave Sine[6] ;
2193:  Track TAST[6] ;
2194:L P[970] WELD_SPEED FINE
    :  Arc End[6]    ;
2195:  Weave End ;
2196:  Track End ;
2197:   ;
 899:   ;
 900:L P[410] 1000mm/sec CNT25    ;
 901:   ;
 902:L P[411] 1200mm/sec CNT40    ;
 903:   ;
 904:  !********POSITIONER MOVE******** ;
 905:J P[412] 90% CNT30    ;
 906:   ;
 907:L P[413] 1000mm/sec CNT25    ;
 908:   ;
 909:L P[414] 1000mm/sec CNT25    ;
 910:   ;
 911:   ;
 912:  !FR50L1610 ;
 913:  IF R[15:TECH HOLD]=1612,CALL TECH_HOLD ;
 914:   ;
 915:   ;
2199:   ;
2200:L P[971] 1000mm/sec FINE
    :  Arc Start[6]    ;
2201:  Weave Sine[6] ;
2202:  Track TAST[6] ;
2203:L P[972] WELD_SPEED CNT100    ;
2204:L P[973] WELD_SPEED FINE
    :  Arc End[6]    ;
2205:  Weave End ;
2206:  Track End ;
2207:   ;
 917:   ;
 918:L P[418] 1000mm/sec CNT25    ;
 919:   ;
 920:L P[419] 1000mm/sec CNT25    ;
 921:   ;
 922:   ;
 923:   ;
 924:  !FR50L1620 ;
 925:  IF R[15:TECH HOLD]=1622,CALL TECH_HOLD ;
 926:   ;
 927:   ;
2209:   ;
2210:L P[974] 1000mm/sec FINE
    :  Arc Start[6]    ;
2211:  Weave Sine[6] ;
2212:  Track TAST[6] ;
2213:L P[975] WELD_SPEED CNT100    ;
2214:L P[976] WELD_SPEED FINE
    :  Arc End[6]    ;
2215:  Weave End ;
2216:  Track End ;
2217:   ;
 929:   ;
 930:L P[423] 1000mm/sec CNT75    ;
 931:   ;
 932:L P[330] 1000mm/sec CNT25    ;
 933:   ;
 934:J P[424] 50% CNT25    ;
 935:   ;
 936:  !********POSITIONER MOVE******** ;
 937:J P[425] 90% CNT30    ;
 938:   ;
 939:J P[426] 50% CNT25    ;
 940:   ;
 941:   ;
 942:  !FR50L1630 ;
 943:  IF R[15:TECH HOLD]=1632,CALL TECH_HOLD ;
 944:   ;
 945:   ;
2219:   ;
2220:L P[977] 1000mm/sec FINE
    :  Arc Start[6]    ;
2221:  Weave Sine[6] ;
2222:  Track TAST[6] ;
2223:L P[978] WELD_SPEED CNT100    ;
2224:C P[979]
    :  P[980] WELD_SPEED CNT100    ;
2225:L P[981] WELD_SPEED CNT100    ;
2226:C P[982]
    :  P[983] WELD_SPEED CNT100    ;
2227:L P[984] WELD_SPEED FINE
    :  Arc End[6]    ;
2228:  Weave End ;
2229:  Track End ;
2230:   ;
 947:   ;
 948:L P[435] 1000mm/sec CNT40    ;
 949:   ;
 950:J P[436] 50% CNT35    ;
 951:   ;
 952:   ;
 953:  !FR50L1640 ;
 954:  IF R[15:TECH HOLD]=1642,CALL TECH_HOLD ;
 955:   ;
 956:   ;
2232:   ;
2233:L P[985] 1000mm/sec FINE
    :  Arc Start[6]    ;
2234:  Weave Sine[6] ;
2235:  Track TAST[6] ;
2236:L P[986] WELD_SPEED CNT100    ;
2237:C P[987]
    :  P[988] WELD_SPEED CNT100    ;
2238:L P[989] WELD_SPEED CNT100    ;
2239:L P[990] WELD_SPEED CNT100    ;
2240:L P[991] WELD_SPEED CNT100    ;
2241:L P[992] WELD_SPEED CNT100    ;
2242:L P[993] WELD_SPEED FINE
    :  Arc End[6]    ;
2243:  Weave End ;
2244:  Track End ;
2245:   ;
 958:   ;
 959:L P[446] 1000mm/sec CNT100    ;
 960:   ;
 961:J P[447] 50% CNT25    ;
 962:   ;
 963:  !********POSITIONER MOVE******** ;
 964:J P[448] 100% FINE    ;
 965:   ;
 966:L P[449] 1000mm/sec CNT25    ;
 967:   ;
 968:J P[450] 50% CNT25    ;
 969:   ;
 970:   ;
 971:  !FR50L1650 ;
 972:  IF R[15:TECH HOLD]=1652,CALL TECH_HOLD ;
 973:   ;
 974:   ;
2247:   ;
2248:L P[994] 1000mm/sec FINE
    :  Arc Start[6]    ;
2249:  Weave Sine[6] ;
2250:L P[995] WELD_SPEED CNT100    ;
2251:L P[996] WELD_SPEED CNT100    ;
2252:L P[997] WELD_SPEED CNT100    ;
2253:  Track TAST[6] ;
2254:L P[998] WELD_SPEED CNT100    ;
2255:L P[999] WELD_SPEED CNT100    ;
2256:L P[1000] WELD_SPEED CNT100    ;
2257:L P[1001] WELD_SPEED CNT100    ;
2258:C P[1002]
    :  P[1003] WELD_SPEED CNT100    ;
2259:L P[1004] WELD_SPEED CNT100    ;
2260:C P[1005]
    :  P[1006] WELD_SPEED CNT100    ;
2261:L P[1007] WELD_SPEED FINE
    :  Arc End[6]    ;
2262:  Weave End ;
2263:  Track End ;
2264:   ;
 976:   ;
 977:L P[465] 1000mm/sec CNT100    ;
 978:   ;
 979:L P[466] 1000mm/sec CNT80    ;
 980:   ;
 981:   ;
 982:  !FR50L1651 ;
 983:  IF R[15:TECH HOLD]=1653,CALL TECH_HOLD ;
 984:   ;
 985:   ;
2266:   ;
2267:L P[1008] 1000mm/sec FINE
    :  Arc Start[6]    ;
2268:  Weave Sine[6] ;
2269:  Track TAST[6] ;
2270:L P[1009] WELD_SPEED CNT100    ;
2271:C P[1010]
    :  P[1011] WELD_SPEED CNT100    ;
2272:C P[1012]
    :  P[1013] WELD_SPEED FINE
    :  Arc End[6]    ;
2273:  Weave End ;
2274:  Track End ;
2275:   ;
 987:   ;
 988:L P[473] 1000mm/sec CNT25    ;
 989:   ;
 990:L P[474] 1000mm/sec CNT100    ;
 991:   ;
 992:L P[475] 1000mm/sec CNT30    ;
 993:   ;
 994:  !HOME ;
 995:J P[88] 100% CNT30    ;
 996:   ;
 997:  !********POSITIONER MOVE******** ;
 998:J P[477] 100% CNT30    ;
 999:   ;
1000:J P[478] 50% CNT100    ;
1001:   ;
1002:J P[479] 50% CNT60    ;
1003:   ;
1004:L P[480] 1000mm/sec CNT25    ;
1005:   ;
1006:   ;
1007:  !FR50L1660 ;
1008:  IF R[15:TECH HOLD]=1662,CALL TECH_HOLD ;
1009:   ;
1010:   ;
2277:   ;
2278:L P[1014] 1000mm/sec FINE
    :  Arc Start[6]    ;
2279:  Weave Sine[6] ;
2280:  Track TAST[6] ;
2281:L P[1015] WELD_SPEED FINE
    :  Arc End[6]    ;
2282:  Weave End ;
2283:  Track End ;
2284:   ;
1012:   ;
1013:J P[483] 20% CNT100    ;
1014:   ;
1015:J P[484] 60% CNT25    ;
1016:   ;
1017:L P[485] 600mm/sec CNT25    ;
1018:   ;
1019:   ;
1020:  !FR50L1661 ;
1021:  IF R[15:TECH HOLD]=1663,CALL TECH_HOLD ;
1022:   ;
1023:   ;
2286:   ;
2287:L P[1016] 1000mm/sec FINE
    :  Arc Start[6]    ;
2288:  Weave Sine[6] ;
2289:  Track TAST[6] ;
2290:L P[1017] WELD_SPEED FINE
    :  Arc End[6]    ;
2291:  Weave End ;
2292:  Track End ;
2293:   ;
1025:   ;
1026:L P[488] 500mm/sec CNT25    ;
1027:   ;
1028:L P[489] 500mm/sec CNT25    ;
1029:   ;
1030:L P[490] 1000mm/sec CNT25    ;
1031:   ;
1032:  !********POSITIONER MOVE******** ;
1033:J P[491] 90% CNT25    ;
1034:   ;
1035:L P[492] 1000mm/sec CNT25    ;
1036:   ;
1037:   ;
1038:  !FR50L1670 ;
1039:  IF R[15:TECH HOLD]=1672,CALL TECH_HOLD ;
1040:   ;
1041:   ;
2295:   ;
2296:L P[1018] 1000mm/sec FINE
    :  Arc Start[8]    ;
2297:  Weave Sine[8] ;
2298:L P[1019] WELD_SPEED FINE
    :  Arc End[8]    ;
2299:  Weave End ;
2300:   ;
1043:   ;
1044:L P[495] 500mm/sec CNT25    ;
1045:   ;
1046:L P[496] 1000mm/sec CNT25    ;
1047:   ;
1048:   ;
1049:  !FR50L1680 ;
1050:  IF R[15:TECH HOLD]=1682,CALL TECH_HOLD ;
1051:   ;
1052:   ;
2302:   ;
2303:L P[1020] 1000mm/sec FINE
    :  Arc Start[6]    ;
2304:  Weave Sine[6] ;
2305:  Track TAST[6] ;
2306:L P[1021] WELD_SPEED FINE
    :  Arc End[6]    ;
2307:  Weave End ;
2308:  Track End ;
2309:   ;
1054:   ;
1055:L P[499] 1000mm/sec CNT25    ;
1056:   ;
1057:  !********POSITIONER MOVE******** ;
1058:J P[500] 75% FINE    ;
1059:   ;
1060:L P[501] 1000mm/sec CNT25    ;
1061:   ;
1062:   ;
1063:  !FR50L1690 ;
1064:  IF R[15:TECH HOLD]=1692,CALL TECH_HOLD ;
1065:   ;
1066:   ;
2311:   ;
2312:L P[1022] 1000mm/sec FINE
    :  Arc Start[6]    ;
2313:  Weave Sine[6] ;
2314:  Track TAST[6] ;
2315:L P[1023] WELD_SPEED CNT100    ;
2316:L P[1024] WELD_SPEED FINE
    :  Arc End[6]    ;
2317:  Weave End ;
2318:  Track End ;
2319:   ;
1068:   ;
1069:L P[505] 300mm/sec CNT25    ;
1070:   ;
1071:L P[506] 1000mm/sec CNT25    ;
1072:   ;
1073:L P[507] 1000mm/sec CNT25    ;
1074:   ;
1075:   ;
1076:  !FR50L1700 ;
1077:  IF R[15:TECH HOLD]=1702,CALL TECH_HOLD ;
1078:   ;
1079:   ;
2321:   ;
2322:L P[1025] 1000mm/sec FINE
    :  Arc Start[6]    ;
2323:  Weave Sine[6] ;
2324:  Track TAST[6] ;
2325:L P[1026] WELD_SPEED CNT100    ;
2326:C P[1027]
    :  P[1028] WELD_SPEED CNT100    ;
2327:L P[1029] WELD_SPEED CNT100    ;
2328:C P[1030]
    :  P[1031] WELD_SPEED CNT100    ;
2329:L P[1032] WELD_SPEED CNT100    ;
2330:C P[1033]
    :  P[1034] WELD_SPEED CNT100    ;
2331:L P[1035] WELD_SPEED FINE
    :  Arc End[6]    ;
2332:  Weave End ;
2333:  Track End ;
2334:   ;
1081:   ;
1082:L P[519] 1000mm/sec CNT100    ;
1083:   ;
1084:L P[520] 1000mm/sec CNT25    ;
1085:   ;
1086:L P[521] 500mm/sec CNT25    ;
1087:   ;
1088:   ;
1089:  !FR50L1710 ;
1090:  IF R[15:TECH HOLD]=1712,CALL TECH_HOLD ;
1091:   ;
1092:   ;
2336:   ;
2337:L P[1036] 1000mm/sec FINE
    :  Arc Start[6]    ;
2338:  Weave Sine[6] ;
2339:  Track TAST[6] ;
2340:L P[1037] WELD_SPEED CNT100    ;
2341:L P[1038] WELD_SPEED FINE
    :  Arc End[6]    ;
2342:  Weave End ;
2343:  Track End ;
2344:   ;
1094:   ;
1095:L P[525] 500mm/sec CNT25    ;
1096:   ;
1097:L P[526] 800mm/sec CNT25    ;
1098:   ;
1099:L P[527] 1000mm/sec CNT100    ;
1100:   ;
1101:J P[528] 50% CNT100    ;
1102:   ;
1103:L P[529] 1000mm/sec CNT25    ;
1104:   ;
1105:   ;
1106:  !FR50L1720 ;
1107:  IF R[15:TECH HOLD]=1722,CALL TECH_HOLD ;
1108:   ;
1109:   ;
2346:   ;
2347:L P[1039] 1000mm/sec FINE
    :  Arc Start[6]    ;
2348:  Weave Sine[6] ;
2349:L P[1040] WELD_SPEED CNT100    ;
2350:L P[1041] WELD_SPEED CNT100    ;
2351:L P[1042] WELD_SPEED FINE
    :  Arc End[6]    ;
2352:  Weave End ;
2353:   ;
1111:   ;
1112:J P[534] 50% CNT10    ;
1113:   ;
1114:  !********POSITIONER MOVE******** ;
1115:J P[535] 40% CNT10    ;
1116:   ;
1117:J P[536] 20% CNT5    ;
1118:   ;
1119:L P[537] 1000mm/sec CNT25    ;
1120:   ;
1121:   ;
1122:  !FR50L1730 ;
1123:  IF R[15:TECH HOLD]=1732,CALL TECH_HOLD ;
1124:   ;
1125:   ;
2355:   ;
2356:L P[1043] 1000mm/sec FINE
    :  Arc Start[6]    ;
2357:  Weave Sine[6] ;
2358:  Track TAST[6] ;
2359:L P[1044] WELD_SPEED CNT100    ;
2360:L P[1045] WELD_SPEED CNT100    ;
2361:L P[1046] WELD_SPEED FINE
    :  Arc End[6]    ;
2362:  Weave End ;
2363:  Track End ;
2364:   ;
1127:   ;
1128:L P[542] 1000mm/sec CNT25    ;
1129:   ;
1130:J P[543] 50% CNT10    ;
1131:   ;
1132:  !********POSITIONER MOVE******** ;
1133:J P[544] 80% CNT10    ;
1134:   ;
1135:   ;
1136:  !FR50L1740 ;
1137:  IF R[15:TECH HOLD]=1742,CALL TECH_HOLD ;
1138:   ;
1139:   ;
2366:   ;
2367:L P[1047] 1000mm/sec FINE
    :  Arc Start[6]    ;
2368:  Weave Sine[6] ;
2369:  Track TAST[6] ;
2370:L P[1048] WELD_SPEED FINE
    :  Arc End[6]    ;
2371:  Weave End ;
2372:  Track End ;
2373:   ;
1141:   ;
1142:L P[547] 1000mm/sec CNT25    ;
1143:   ;
1144:L P[548] 1000mm/sec CNT25    ;
1145:   ;
1146:L P[549] 1000mm/sec CNT25    ;
1147:   ;
1148:   ;
1149:  !FR50L1750 ;
1150:  IF R[15:TECH HOLD]=1752,CALL TECH_HOLD ;
1151:   ;
1152:   ;
2375:   ;
2376:L P[1049] 1000mm/sec FINE
    :  Arc Start[6]    ;
2377:  Weave Sine[6] ;
2378:  Track TAST[6] ;
2379:L P[1050] WELD_SPEED CNT100    ;
2380:L P[1051] WELD_SPEED FINE
    :  Arc End[6]    ;
2381:  Weave End ;
2382:  Track End ;
2383:   ;
1154:   ;
1155:L P[553] 1000mm/sec CNT25    ;
1156:   ;
1157:L P[554] 1000mm/sec CNT100    ;
1158:   ;
1159:L P[555] 1000mm/sec CNT100    ;
1160:   ;
1161:L P[556] 1000mm/sec CNT40    ;
1162:   ;
1163:   ;
1164:  !FR50L1770 ;
1165:  IF R[15:TECH HOLD]=1772,CALL TECH_HOLD ;
1166:   ;
1167:   ;
2385:   ;
2386:L P[1052] 1000mm/sec FINE
    :  Arc Start[6]    ;
2387:  Weave Sine[6] ;
2388:  Track TAST[6] ;
2389:L P[1053] WELD_SPEED FINE
    :  Arc End[6]    ;
2390:  Weave End ;
2391:  Track End ;
2392:L P[1054] 1000mm/sec FINE
    :  Arc Start[6]    ;
2393:  Weave Sine[6] ;
2394:L P[1055] WELD_SPEED FINE
    :  Arc End[6]    ;
2395:  Weave End ;
2396:L P[1056] 2400mm/sec FINE
    :  Arc Start[6]    ;
2397:  Weave Sine[6] ;
2398:L P[1057] WELD_SPEED FINE
    :  Arc End[6]    ;
2399:  Weave End ;
2400:   ;
1169:   ;
1170:L P[559] 1000mm/sec CNT100    ;
1171:   ;
1172:L P[560] 1000mm/sec CNT25    ;
1173:   ;
1176:L P[563] 1200mm/sec CNT100    ;
1177:   ;
1178:L P[89] 800mm/sec CNT100    ;
1179:   ;
1180:J P[565] 30% CNT20    ;
1181:   ;
1184:J P[568] 25% CNT25    ;
1185:   ;
1186:J P[569] 50% CNT100    ;
1187:   ;
1188:  !HOME ;
1189:J P[90] 100% CNT30    ;
1190:   ;
1191:  !********POSITIONER MOVE******** ;
1192:J P[570] 100% CNT30    ;
1193:   ;
1194:J P[371] 50% CNT100    ;
1195:   ;
1196:L P[572] 1000mm/sec CNT25    ;
1197:   ;
1198:L P[573] 1000mm/sec CNT25    ;
1199:   ;
1200:   ;
1201:  !FR50L1780 ;
1202:  IF R[15:TECH HOLD]=1782,CALL TECH_HOLD ;
1203:   ;
1204:   ;
2402:   ;
2403:L P[1058] 500mm/sec FINE
    :  Arc Start[6]    ;
2404:  Weave Sine[6] ;
2405:  Track TAST[6] ;
2406:L P[1059] WELD_SPEED FINE
    :  Arc End[6]    ;
2407:  Weave End ;
2408:  Track End ;
2409:   ;
1206:   ;
1207:L P[576] 500mm/sec CNT25    ;
1208:   ;
1209:L P[577] 1000mm/sec CNT25    ;
1210:   ;
1211:  !********POSITIONER MOVE******** ;
1212:J P[578] 100% FINE    ;
1213:   ;
1214:   ;
1215:  !FR50L1790 ;
1216:  IF R[15:TECH HOLD]=1792,CALL TECH_HOLD ;
1217:   ;
1218:   ;
2411:   ;
2412:L P[1060] 1000mm/sec FINE
    :  Arc Start[6]    ;
2413:  Weave Sine[6] ;
2414:  Track TAST[6] ;
2415:L P[1061] WELD_SPEED FINE
    :  Arc End[6]    ;
2416:  Weave End ;
2417:  Track End ;
2418:   ;
1220:   ;
1221:L P[581] 1000mm/sec CNT100    ;
1222:   ;
1223:   ;
1224:  !FR50L1800 ;
1225:  IF R[15:TECH HOLD]=1802,CALL TECH_HOLD ;
1226:   ;
1227:   ;
2420:   ;
2421:L P[1062] 1000mm/sec FINE
    :  Arc Start[6]    ;
2422:  Weave Sine[6] ;
2423:  Track TAST[6] ;
2424:L P[1063] WELD_SPEED CNT100    ;
2425:L P[1064] WELD_SPEED FINE
    :  Arc End[6]    ;
2426:  Weave End ;
2427:  Track End ;
2428:   ;
1229:   ;
1230:L P[585] 1000mm/sec CNT25    ;
1231:   ;
1232:   ;
1233:  !FR50L1810 ;
1234:  IF R[15:TECH HOLD]=1812,CALL TECH_HOLD ;
1235:   ;
1236:   ;
2430:   ;
2431:L P[1065] 1000mm/sec FINE
    :  Arc Start[6]    ;
2432:  Weave Sine[6] ;
2433:  Track TAST[6] ;
2434:L P[1066] WELD_SPEED CNT100    ;
2435:L P[1067] WELD_SPEED FINE
    :  Arc End[6]    ;
2436:  Weave End ;
2437:  Track End ;
2438:   ;
1238:   ;
1239:L P[589] 1000mm/sec CNT25    ;
1240:   ;
1241:J P[590] 50% CNT25    ;
1242:   ;
1243:L P[591] 1000mm/sec CNT25    ;
1244:   ;
1245:   ;
1246:  !FR50L1820 ;
1247:  IF R[15:TECH HOLD]=1822,CALL TECH_HOLD ;
1248:   ;
1249:   ;
2440:   ;
2441:L P[1068] 1000mm/sec FINE
    :  Arc Start[6]    ;
2442:  Weave Sine[6] ;
2443:L P[1069] WELD_SPEED CNT100    ;
2444:L P[1070] WELD_SPEED FINE
    :  Arc End[6]    ;
2445:  Weave End ;
2446:   ;
1251:   ;
1252:L P[595] 1000mm/sec CNT25    ;
1253:   ;
1254:J P[596] 50% CNT100    ;
1255:   ;
1256:J P[597] 50% CNT100    ;
1257:   ;
1258:L P[598] 1000mm/sec CNT25    ;
1259:   ;
1260:   ;
1261:   ;
1262:  !FR50L1830 ;
1263:  IF R[15:TECH HOLD]=1832,CALL TECH_HOLD ;
1264:   ;
1265:   ;
2448:   ;
2449:L P[1071] 1000mm/sec FINE
    :  Arc Start[6]    ;
2450:  Weave Sine[6] ;
2451:  Track TAST[6] ;
2452:L P[1072] WELD_SPEED CNT100    ;
2453:C P[1073]
    :  P[1074] WELD_SPEED CNT100    ;
2454:L P[1075] WELD_SPEED CNT100    ;
2455:C P[1076]
    :  P[1077] WELD_SPEED CNT100    ;
2456:L P[1078] WELD_SPEED FINE
    :  Arc End[6]    ;
2457:  Weave End ;
2458:  Track End ;
2459:   ;
1267:   ;
1268:L P[607] 1000mm/sec CNT60    ;
1269:   ;
1270:J P[608] 50% CNT50    ;
1271:   ;
1272:   ;
1273:  !FR50L1840 ;
1274:  IF R[15:TECH HOLD]=1842,CALL TECH_HOLD ;
1275:   ;
1276:   ;
2461:   ;
2462:L P[1079] 1000mm/sec FINE
    :  Arc Start[6]    ;
2463:  Weave Sine[6] ;
2464:  Track TAST[6] ;
2465:L P[1080] WELD_SPEED CNT100    ;
2466:C P[1081]
    :  P[1082] WELD_SPEED CNT100    ;
2467:L P[1083] WELD_SPEED CNT100    ;
2468:L P[1084] WELD_SPEED CNT100    ;
2469:L P[1085] WELD_SPEED CNT100    ;
2470:L P[1086] WELD_SPEED CNT100    ;
2471:L P[1087] WELD_SPEED FINE
    :  Arc End[6]    ;
2472:  Weave End ;
2473:  Track End ;
2474:   ;
1278:   ;
1279:L P[618] 1000mm/sec CNT25    ;
1280:   ;
1281:J P[619] 50% CNT100    ;
1282:   ;
1283:J P[620] 50% CNT100    ;
1284:   ;
1285:J P[372] 50% CNT100    ;
1286:   ;
1287:L P[621] 1000mm/sec CNT25    ;
1288:   ;
1289:   ;
1290:  !FR50L1850 ;
1291:  IF R[15:TECH HOLD]=1852,CALL TECH_HOLD ;
1292:   ;
2476:   ;
2477:L P[1088] 1000mm/sec FINE
    :  Arc Start[6]    ;
2478:  Weave Sine[6] ;
2479:L P[1089] WELD_SPEED CNT100    ;
2480:L P[1090] WELD_SPEED CNT100    ;
2481:L P[1091] WELD_SPEED FINE
    :  Arc End[6]    ;
2482:  Weave End ;
2483:   ;
1294:   ;
1295:L P[626] 1000mm/sec CNT100    ;
1296:   ;
1297:L P[627] 1000mm/sec CNT100    ;
1298:   ;
1299:   ;
1300:  !FR50L1860 ;
1301:  IF R[15:TECH HOLD]=1862,CALL TECH_HOLD ;
1302:   ;
1303:   ;
2485:   ;
2486:L P[1092] 1000mm/sec FINE
    :  Arc Start[6]    ;
2487:  Weave Sine[6] ;
2488:  Track TAST[6] ;
2489:L P[1093] WELD_SPEED FINE
    :  Arc End[6]    ;
2490:  Weave End ;
2491:  Track End ;
2492:   ;
1305:   ;
1306:L P[630] 1000mm/sec CNT50    ;
1307:   ;
1308:   ;
1309:  !FR50L1870 ;
1310:  IF R[15:TECH HOLD]=1872,CALL TECH_HOLD ;
1311:   ;
1312:   ;
2494:   ;
2495:L P[1094] 1000mm/sec FINE
    :  Arc Start[6]    ;
2496:  Weave Sine[6] ;
2497:  Track TAST[6] ;
2498:L P[1095] WELD_SPEED CNT100    ;
2499:L P[1096] WELD_SPEED FINE
    :  Arc End[6]    ;
2500:  Weave End ;
2501:  Track End ;
2502:   ;
1314:   ;
1315:L P[634] 1000mm/sec CNT60    ;
1316:   ;
1317:   ;
1318:  !FR50L1880 ;
1319:  IF R[15:TECH HOLD]=1882,CALL TECH_HOLD ;
1320:   ;
1321:   ;
2504:   ;
2505:L P[1097] 1000mm/sec FINE
    :  Arc Start[6]    ;
2506:  Weave Sine[6] ;
2507:  Track TAST[6] ;
2508:L P[1098] WELD_SPEED CNT100    ;
2509:L P[1099] WELD_SPEED FINE
    :  Arc End[6]    ;
2510:  Weave End ;
2511:  Track End ;
2512:   ;
1323:   ;
1324:L P[373] 1000mm/sec CNT25    ;
1325:   ;
1326:J P[638] 50% CNT25    ;
1327:   ;
1328:J P[641] 50% CNT25    ;
1329:   ;
1330:   ;
1331:  !FR50L1900 ;
1332:  IF R[15:TECH HOLD]=1902,CALL TECH_HOLD ;
1333:   ;
1334:   ;
2514:   ;
2515:L P[1100] 1000mm/sec FINE
    :  Arc Start[6]    ;
2516:  Weave Sine[6] ;
2517:  Track TAST[6] ;
2518:L P[1101] WELD_SPEED CNT100    ;
2519:L P[1102] WELD_SPEED FINE
    :  Arc End[6]    ;
2520:  Weave End ;
2521:  Track End ;
2522:   ;
1336:   ;
1337:L P[645] 1000mm/sec CNT25    ;
1338:   ;
1339:  !********POSITIONER MOVE******** ;
1340:J P[646] 100% FINE    ;
1341:   ;
1342:L P[647] 1000mm/sec CNT25    ;
1343:   ;
1344:L P[648] 1000mm/sec CNT25    ;
1345:   ;
1346:   ;
1347:  !FR50L1910 ;
1348:  IF R[15:TECH HOLD]=1912,CALL TECH_HOLD ;
1349:   ;
1350:   ;
2524:   ;
2525:L P[1103] 1000mm/sec FINE
    :  Arc Start[6]    ;
2526:  Weave Sine[6] ;
2527:  Track TAST[6] ;
2528:L P[1104] WELD_SPEED CNT100    ;
2529:C P[1105]
    :  P[1106] WELD_SPEED CNT100    ;
2530:L P[1107] WELD_SPEED CNT100    ;
2531:L P[1108] WELD_SPEED CNT100    ;
2532:L P[1109] WELD_SPEED CNT100    ;
2533:L P[1110] WELD_SPEED CNT100    ;
2534:C P[1111]
    :  P[1112] WELD_SPEED CNT100    ;
2535:L P[1113] WELD_SPEED CNT100    ;
2536:C P[1114]
    :  P[1115] WELD_SPEED CNT100    ;
2537:L P[1116] WELD_SPEED CNT100    ;
2538:C P[1117]
    :  P[1118] WELD_SPEED CNT100    ;
2539:L P[1119] WELD_SPEED CNT100    ;
2540:L P[1120] WELD_SPEED CNT100    ;
2541:L P[1121] WELD_SPEED CNT100    ;
2542:C P[1122]
    :  P[1123] WELD_SPEED FINE
    :  Arc End[6]    ;
2543:  Weave End ;
2544:  Track End ;
2545:   ;
2546:  !FR50l1911 ;
2547:   ;
2548:L P[1124] 500mm/sec FINE
    :  Arc Start[6]    ;
2549:  Weave Sine[6] ;
2550:  Track TAST[6] ;
2551:L P[1125] WELD_SPEED CNT100    ;
2552:C P[1126]
    :  P[1127] WELD_SPEED CNT100    ;
2553:L P[1128] WELD_SPEED CNT100    ;
2554:C P[1129]
    :  P[1130] WELD_SPEED FINE
    :  Arc End[6]    ;
2555:  Weave End ;
2556:  Track End ;
2557:   ;
1352:   ;
1353:L P[670] 1000mm/sec CNT25    ;
1354:   ;
1355:L P[671] 500mm/sec CNT25    ;
1356:   ;
1357:   ;
1358:  !FR50L1911 ;
1359:  IF R[15:TECH HOLD]=1913,CALL TECH_HOLD ;
1360:   ;
1361:   ;
1364:L P[679] 1000mm/sec CNT100    ;
1365:   ;
1366:J P[680] 50% CNT100    ;
1367:   ;
1368:J P[95] 50% CNT100    ;
1369:   ;
1370:J P[681] 50% CNT50    ;
1371:   ;
1372:  !HOME ;
1373:J P[94] 100% FINE    ;
1374:   ;
1375:  CALL T_CLEAN    ;
1376:   ;
1377:  !********POSITIONER MOVE******** ;
1378:J P[682] 90% CNT30    ;
1379:   ;
1380:J P[683] 50% CNT25    ;
1381:   ;
1382:J P[684] 50% CNT25    ;
1383:   ;
1384:L P[685] 1000mm/sec CNT25    ;
1385:   ;
1386:  !TO SKIP FRONT BUMPER WELDS ;
1387:  CALL ARC_DISABLE_FRONT_BMPR_LRG(0) ;
1388:   ;
1389:  !FR50L1920 ;
1390:  IF R[15:TECH HOLD]=1922,CALL TECH_HOLD ;
1391:   ;
1392:   ;
2559:   ;
2560:L P[1131] 1000mm/sec FINE
    :  Arc Start[6]    ;
2561:  Weave Sine[6] ;
2562:  Track TAST[6] ;
2563:L P[1132] WELD_SPEED FINE
    :  Arc End[6]    ;
2564:  Weave End ;
2565:  Track End ;
2566:   ;
1394:   ;
1395:L P[688] 1000mm/sec CNT100    ;
1396:   ;
1397:J P[689] 50% CNT25    ;
1398:   ;
1399:L P[690] 1000mm/sec CNT25    ;
1400:   ;
1401:   ;
1402:  !FR50L1930 ;
1403:  IF R[15:TECH HOLD]=1932,CALL TECH_HOLD ;
2568:   ;
2569:L P[1133] 1000mm/sec FINE
    :  Arc Start[6]    ;
2570:  Weave Sine[6] ;
2571:  Track TAST[6] ;
2572:L P[1134] WELD_SPEED CNT100    ;
2573:L P[1135] WELD_SPEED FINE
    :  Arc End[6]    ;
2574:  Weave End ;
2575:  Track End ;
2576:   ;
1405:   ;
1406:L P[694] 1000mm/sec CNT100    ;
1407:   ;
1408:L P[695] 1000mm/sec CNT100    ;
1409:   ;
1410:  !FR50L1940 ;
1411:  IF R[15:TECH HOLD]=1942,CALL TECH_HOLD ;
1412:   ;
1413:   ;
2578:   ;
2579:L P[1136] 1000mm/sec FINE
    :  Arc Start[6]    ;
2580:  Weave Sine[6] ;
2581:  Track TAST[6] ;
2582:L P[1137] WELD_SPEED FINE
    :  Arc End[6]    ;
2583:  Weave End ;
2584:  Track End ;
2585:   ;
1415:   ;
1416:  CALL ARC_DISABLE_FRONT_BMPR_LRG(1) ;
1417:   ;
1418:L P[698] 1000mm/sec CNT25    ;
1419:   ;
1420:J P[699] 70% CNT40    ;
1421:   ;
1422:  !********POSITIONER MOVE******** ;
1423:J P[700] 90% CNT30    ;
1424:   ;
1425:L P[701] 1000mm/sec CNT25    ;
1426:   ;
1427:   ;
1428:  CALL ARC_ENABLE_LH_LS(0) ;
1429:   ;
1430:  !FR50L1950 ;
1431:  IF R[15:TECH HOLD]=1952,CALL TECH_HOLD ;
1432:   ;
1433:   ;
1434:L P[702] 1000mm/sec CNT25    ;
1435:   ;
2587:   ;
2588:L P[1138] 1000mm/sec FINE
    :  Arc Start[6]    ;
2589:  Weave Sine[6] ;
2590:  Track TAST[6] ;
2591:L P[1139] WELD_SPEED CNT100    ;
2592:L P[1140] WELD_SPEED CNT100    ;
2593:C P[1141]
    :  P[1142] WELD_SPEED FINE
    :  Arc End[6]    ;
2594:  Weave End ;
2595:  Track End ;
2596:   ;
1437:   ;
1438:  CALL ARC_ENABLE_LH_LS(1) ;
1439:   ;
1440:L P[708] 1000mm/sec CNT50    ;
1441:   ;
1442:J P[97] 50% CNT25    ;
1443:   ;
1444:J P[710] 50% CNT25    ;
1445:   ;
1446:  !HOME ;
1447:J P[98] 100% CNT50    ;
1448:   ;
1449:  !********POSITIONER MOVE******** ;
1450:J P[2] 85% CNT100    ;
1451:   ;
1452:J P[105] 50% CNT25    ;
1453:   ;
1454:L P[113] 1000mm/sec CNT25    ;
1455:   ;
1456:  CALL ARC_ENABLE_RH_LS(0) ;
1457:   ;
1458:  !FR50L1970 ;
1459:  IF R[15:TECH HOLD]=1972,CALL TECH_HOLD ;
1460:   ;
1461:   ;
2609:   ;
2610:L P[1148] 800mm/sec FINE
    :  Arc Start[6]    ;
2611:  Weave Sine[6] ;
2612:  Track TAST[6] ;
2613:L P[1149] WELD_SPEED CNT100    ;
2614:C P[1150]
    :  P[1151] WELD_SPEED FINE
    :  Arc End[6]    ;
2615:  Track End ;
2616:  Weave End ;
2617:   ;
1463:   ;
1464:L P[564] 800mm/sec CNT5    ;
1465:   ;
1466:J P[571] 20% CNT40    ;
1467:   ;
1468:J P[639] 40% CNT25    ;
1469:   ;
1470:J P[640] 75% CNT50    ;
1471:   ;
1472:  !********POSITIONER MOVE******** ;
1473:J P[711] 85% CNT30    ;
1474:   ;
1475:J P[712] 50% CNT100    ;
1476:   ;
1477:L P[713] 1000mm/sec CNT25    ;
1478:   ;
1479:   ;
1480:  !FR50L1960 ;
1481:  IF R[15:TECH HOLD]=1962,CALL TECH_HOLD ;
1482:   ;
1483:   ;
1484:L P[714] 500mm/sec CNT25    ;
1485:   ;
2598:   ;
2599:L P[1143] 1000mm/sec FINE
    :  Arc Start[6]    ;
2600:  Weave Sine[6] ;
2601:  Track TAST[6] ;
2602:L P[1144] WELD_SPEED CNT100    ;
2603:L P[1145] WELD_SPEED CNT100    ;
2604:C P[1146]
    :  P[1147] WELD_SPEED FINE
    :  Arc End[6]    ;
2605:  Weave End ;
2606:  Track End ;
2607:   ;
1487:   ;
1488:  CALL ARC_ENABLE_RH_LS(1) ;
1489:   ;
1490:L P[720] 500mm/sec CNT25    ;
1491:   ;
1492:L P[721] 1000mm/sec CNT100    ;
1493:   ;
1494:J P[99] 100% CNT30    ;
1495:   ;
1496:  !******** POSITIONER MOVE ******* ;
1497:J P[793] 85% CNT30    ;
1498:   ;
1499:J P[732] 75% CNT25    ;
1500:   ;
1501:L P[733] 1000mm/sec CNT100    ;
1502:   ;
1503:   ;
1504:  CALL ARC_ENABLE_LH_LS(0) ;
1505:   ;
1506:  !FR50L1980 ;
1507:  IF R[15:TECH HOLD]=1982,CALL TECH_HOLD ;
1508:   ;
1509:   ;
2619:   ;
2620:L P[1152] 800mm/sec FINE
    :  Arc Start[6]    ;
2621:  Weave Sine[6] ;
2622:  Track TAST[6] ;
2623:L P[1153] WELD_SPEED CNT100    ;
2624:C P[1154]
    :  P[1155] WELD_SPEED FINE
    :  Arc End[6]    ;
2625:  Weave End ;
2626:  Track End ;
2627:   ;
2628:   ;
1511:   ;
1512:L P[738] 800mm/sec CNT20    ;
1513:   ;
1514:L P[739] 1000mm/sec CNT100    ;
1515:   ;
1516:J P[740] 100% CNT100    ;
1517:   ;
1518:  !HOME ;
1519:J P[104] 100% CNT30    ;
1520:   ;
1521:   ;
1522:  !********POSITIONER MOVE******** ;
1523:J P[722] 85% CNT30    ;
1524:   ;
1525:J P[106] 50% CNT90    ;
1526:   ;
1527:   ;
1528:  !FR50L2010 ;
1529:  IF R[15:TECH HOLD]=2012,CALL TECH_HOLD ;
1530:   ;
1531:L P[756] 1000mm/sec CNT25    ;
1532:   ;
2630:   ;
2631:L P[1162] 1000mm/sec FINE
    :  Arc Start[8]    ;
2632:  Weave Sine[8] ;
2633:L P[1163] WELD_SPEED CNT100    ;
2634:C P[1164]
    :  P[1165] WELD_SPEED CNT100    ;
2635:L P[1166] WELD_SPEED CNT100    ;
2636:L P[1167] WELD_SPEED CNT100    ;
2637:L P[1168] WELD_SPEED CNT100    ;
2638:L P[1169] WELD_SPEED FINE
    :  Arc End[8]    ;
2639:  Weave End ;
2640:   ;
1534:   ;
1535:  CALL ARC_ENABLE_LH_LS(1) ;
1536:   ;
1537:L P[765] 1000mm/sec CNT50    ;
1538:   ;
1539:J P[109] 50% CNT100    ;
1540:   ;
1541:J P[108] 50% CNT70    ;
1542:   ;
1543:  !HOME ;
1544:J P[107] 100% CNT50    ;
1545:   ;
1546:   ;
1547:  !********POSITIONER MOVE******** ;
1548:J P[778] 90% CNT30    ;
1549:   ;
1550:J P[780] 50% CNT25    ;
1551:   ;
1552:  CALL ARC_ENABLE_RH_LS(0) ;
1553:   ;
1554:   ;
1555:  !FR50L2040 ;
1556:  IF R[15:TECH HOLD]=2042,CALL TECH_HOLD ;
1557:   ;
1558:   ;
1559:L P[781] 1000mm/sec CNT25    ;
1560:   ;
1563:  CALL ARC_ENABLE_RH_LS(1) ;
1564:   ;
1565:L P[790] 1000mm/sec CNT25    ;
1566:   ;
1567:J P[115] 50% CNT100    ;
1568:   ;
1569:  !HOME ;
1570:J P[114] 100% CNT10    ;
1571:  CALL HOME    ;
1572:   ;
1573:  !********POSITIONER MOVE******** ;
1574:  CALL LOAD_POS    ;
1575:   ;
/POS
P[1]{
   GP1:
	UF : 1, UT : 1,		CONFIG : 'N U T, 0, 0, 0',
	X =  1048.285  mm,	Y = -1294.070  mm,	Z =   701.250  mm,
	W =     -.009 deg,	P =    41.863 deg,	R =  -150.867 deg
   GP2:
	UF : 1, UT : 1,
	J1=     0.000 deg,	J2=   -40.000 deg
};
P[2]{
   GP1:
	UF : 1, UT : 1,		CONFIG : 'N U T, 0, 0, 0',
	X =  1163.054  mm,	Y = -1078.949  mm,	Z =  1751.193  mm,
	W =   -29.332 deg,	P =   -12.370 deg,	R =    13.560 deg
   GP2:
	UF : 1, UT : 1,
	J1=   180.000 deg,	J2=  -125.000 deg
};
P[3]{
   GP1:
	UF : 1, UT : 1,		CONFIG : 'N U T, 0, 0, 0',
	X =  1209.555  mm,	Y = -1322.972  mm,	Z =   229.179  mm,
	W =     -.010 deg,	P =    41.970 deg,	R =  -145.526 deg
   GP2:
	UF : 1, UT : 1,
	J1=     0.000 deg,	J2=   -40.000 deg
};
P[4]{
   GP1:
	UF : 1, UT : 1,		CONFIG : 'N U B, 0, 0, 0',
	X =   356.032  mm,	Y =    -2.146  mm,	Z =  2424.050  mm,
	W =      .001 deg,	P =   -40.002 deg,	R =     -.005 deg
   GP2:
	UF : 1, UT : 1,
	J1=     0.000 deg,	J2=   -40.000 deg
};
P[5]{
   GP1:
	UF : 1, UT : 1,		CONFIG : 'N U T, 0, 0, 0',
	X =  1269.879  mm,	Y = -1253.433  mm,	Z =    79.373  mm,
	W =    -1.683 deg,	P =    44.139 deg,	R =  -145.609 deg
   GP2:
	UF : 1, UT : 1,
	J1=     0.000 deg,	J2=   -40.000 deg
};
P[6]{
   GP1:
	UF : 1, UT : 1,		CONFIG : 'N U T, 0, 0, 0',
	X =  1314.620  mm,	Y = -1313.270  mm,	Z =    82.919  mm,
	W =     1.498 deg,	P =    44.726 deg,	R =  -177.480 deg
   GP2:
	UF : 1, UT : 1,
	J1=     0.000 deg,	J2=   -40.000 deg
};
P[7]{
   GP1:
	UF : 1, UT : 1,		CONFIG : 'N U B, 0, 0, 0',
	X =   356.032  mm,	Y =    -2.146  mm,	Z =  2424.049  mm,
	W =      .001 deg,	P =   -40.002 deg,	R =     -.005 deg
   GP2:
	UF : 1, UT : 1,
	J1=    45.000 deg,	J2=     0.000 deg
};
P[8]{
   GP1:
	UF : 1, UT : 1,		CONFIG : 'N U T, 0, 0, 0',
	X =  1272.049  mm,	Y = -1319.952  mm,	Z =   170.275  mm,
	W =    -4.003 deg,	P =    44.859 deg,	R =  -166.486 deg
   GP2:
	UF : 1, UT : 1,
	J1=     0.000 deg,	J2=   -40.000 deg
};
P[9]{
   GP1:
	UF : 1, UT : 1,		CONFIG : 'N U T, 0, 0, 0',
	X =   909.960  mm,	Y =  -872.839  mm,	Z =   170.274  mm,
	W =      .297 deg,	P =    44.999 deg,	R =  -138.174 deg
   GP2:
	UF : 1, UT : 1,
	J1=     0.000 deg,	J2=   -40.000 deg
};
P[10]{
   GP1:
	UF : 1, UT : 1,		CONFIG : 'N U T, 0, 0, 0',
	X =   907.923  mm,	Y =  -828.465  mm,	Z =    78.992  mm,
	W =     -.234 deg,	P =    44.187 deg,	R =  -138.544 deg
   GP2:
	UF : 1, UT : 1,
	J1=     0.000 deg,	J2=   -40.000 deg
};
P[11]{
   GP1:
	UF : 1, UT : 1,		CONFIG : 'N U T, 0, 0, 0',
	X =  1239.992  mm,	Y = -1224.689  mm,	Z =    81.310  mm,
	W =      .993 deg,	P =    44.648 deg,	R =  -147.123 deg
   GP2:
	UF : 1, UT : 1,
	J1=     0.000 deg,	J2=   -40.000 deg
};
P[12]{
   GP1:
	UF : 1, UT : 1,		CONFIG : 'N U T, 0, 0, 0',
	X =  1163.391  mm,	Y = -1298.112  mm,	Z =   230.228  mm,
	W =     1.291 deg,	P =    44.986 deg,	R =  -138.174 deg
   GP2:
	UF : 1, UT : 1,
	J1=     0.000 deg,	J2=   -40.000 deg
};
P[13]{
   GP1:
	UF : 1, UT : 1,		CONFIG : 'N U T, 0, 0, 0',
	X =   860.828  mm,	Y =  -857.112  mm,	Z =   230.228  mm,
	W =     1.291 deg,	P =    44.986 deg,	R =  -138.174 deg
   GP2:
	UF : 1, UT : 1,
	J1=     0.000 deg,	J2=   -40.000 deg
};
P[14]{
   GP1:
	UF : 1, UT : 1,		CONFIG : 'N U T, 0, 0, 0',
	X =   882.027  mm,	Y =  -793.098  mm,	Z =    83.021  mm,
	W =    -1.714 deg,	P =    41.650 deg,	R =  -137.126 deg
   GP2:
	UF : 1, UT : 1,
	J1=     0.000 deg,	J2=   -40.000 deg
};
P[15]{
   GP1:
	UF : 1, UT : 1,		CONFIG : 'N U T, 0, 0, 0',
	X =   833.656  mm,	Y =  -734.388  mm,	Z =    84.663  mm,
	W =    -1.870 deg,	P =    41.238 deg,	R =  -117.739 deg
   GP2:
	UF : 1, UT : 1,
	J1=     0.000 deg,	J2=   -40.000 deg
};
P[16]{
   GP1:
	UF : 1, UT : 1,		CONFIG : 'N U T, 0, 0, 0',
	X =   643.854  mm,	Y = -1045.560  mm,	Z =   456.782  mm,
	W =     1.290 deg,	P =    44.986 deg,	R =  -124.491 deg
   GP2:
	UF : 1, UT : 1,
	J1=     0.000 deg,	J2=   -40.000 deg
};
P[17]{
   GP1:
	UF : 1, UT : 1,		CONFIG : 'N U T, 0, 0, 0',
	X =   908.243  mm,	Y =     -.972  mm,	Z =  2177.323  mm,
	W =     -.010 deg,	P =   -45.000 deg,	R =     0.000 deg
   GP2:
	UF : 1, UT : 1,
	J1=    90.000 deg,	J2=     0.000 deg
};
P[18]{
   GP1:
	UF : 1, UT : 1,		CONFIG : 'N U T, 0, 0, 0',
	X =  1593.884  mm,	Y =    54.651  mm,	Z =  1425.564  mm,
	W =    40.560 deg,	P =     2.984 deg,	R =   -28.829 deg
   GP2:
	UF : 1, UT : 1,
	J1=    90.000 deg,	J2=     0.000 deg
};
P[19]{
   GP1:
	UF : 1, UT : 1,		CONFIG : 'N U T, 0, 0, 0',
	X =  2419.244  mm,	Y =   170.457  mm,	Z =   756.322  mm,
	W =    40.554 deg,	P =     2.977 deg,	R =   -28.823 deg
   GP2:
	UF : 1, UT : 1,
	J1=    90.000 deg,	J2=     0.000 deg
};
P[20]{
   GP1:
	UF : 1, UT : 1,		CONFIG : 'N U T, 0, 0, 0',
	X =  2486.244  mm,	Y =   320.457  mm,	Z =   579.520  mm,
	W =    40.554 deg,	P =     2.977 deg,	R =    -7.352 deg
   GP2:
	UF : 1, UT : 1,
	J1=    90.000 deg,	J2=     0.000 deg
};
P[21]{
   GP1:
	UF : 1, UT : 1,		CONFIG : 'N U T, 0, 0, 0',
	X =  2507.432  mm,	Y =   427.190  mm,	Z =   497.403  mm,
	W =    44.780 deg,	P =     5.017 deg,	R =    -1.188 deg
   GP2:
	UF : 1, UT : 1,
	J1=    90.000 deg,	J2=     0.000 deg
};
P[22]{
   GP1:
	UF : 1, UT : 1,		CONFIG : 'N U T, 0, 0, 0',
	X =  2456.052  mm,	Y =   425.683  mm,	Z =   498.220  mm,
	W =    45.076 deg,	P =     5.046 deg,	R =    -1.313 deg
   GP2:
	UF : 1, UT : 1,
	J1=    89.999 deg,	J2=     0.000 deg
};
P[23]{
   GP1:
	UF : 1, UT : 1,		CONFIG : 'N U T, 0, 0, 0',
	X =  2440.584  mm,	Y =   427.227  mm,	Z =   496.365  mm,
	W =    44.794 deg,	P =     5.016 deg,	R =    30.070 deg
   GP2:
	UF : 1, UT : 1,
	J1=    90.000 deg,	J2=     0.000 deg
};
P[24]{
   GP1:
	UF : 1, UT : 1,		CONFIG : 'N U T, 0, 0, 0',
	X =  2521.819  mm,	Y =   261.320  mm,	Z =   656.993  mm,
	W =    44.759 deg,	P =     5.240 deg,	R =    21.047 deg
   GP2:
	UF : 1, UT : 1,
	J1=    90.000 deg,	J2=     0.000 deg
};
P[25]{
   GP1:
	UF : 1, UT : 1,		CONFIG : 'N U T, 0, 0, 0',
	X =  2511.367  mm,	Y =  -251.873  mm,	Z =   577.119  mm,
	W =   -39.345 deg,	P =     9.413 deg,	R =    11.283 deg
   GP2:
	UF : 1, UT : 1,
	J1=    90.000 deg,	J2=     0.000 deg
};
P[26]{
   GP1:
	UF : 1, UT : 1,		CONFIG : 'N U T, 0, 0, 0',
	X =  2524.023  mm,	Y =  -405.057  mm,	Z =   494.826  mm,
	W =   -44.056 deg,	P =    10.309 deg,	R =     9.167 deg
   GP2:
	UF : 1, UT : 1,
	J1=    90.000 deg,	J2=     0.000 deg
};
P[27]{
   GP1:
	UF : 1, UT : 1,		CONFIG : 'N U T, 0, 0, 0',
	X =  2485.759  mm,	Y =  -405.522  mm,	Z =   494.261  mm,
	W =   -44.059 deg,	P =    10.320 deg,	R =     9.160 deg
   GP2:
	UF : 1, UT : 1,
	J1=    90.000 deg,	J2=     0.000 deg
};
P[28]{
   GP1:
	UF : 1, UT : 1,		CONFIG : 'N U T, 0, 0, 0',
	X =  2449.237  mm,	Y =  -403.696  mm,	Z =   493.863  mm,
	W =   -44.053 deg,	P =    10.305 deg,	R =   -21.685 deg
   GP2:
	UF : 1, UT : 1,
	J1=    90.000 deg,	J2=     0.000 deg
};
P[29]{
   GP1:
	UF : 1, UT : 1,		CONFIG : 'N U T, 0, 0, 0',
	X =  2549.787  mm,	Y =  -262.671  mm,	Z =   682.477  mm,
	W =   -44.052 deg,	P =    10.305 deg,	R =   -20.066 deg
   GP2:
	UF : 1, UT : 1,
	J1=    90.000 deg,	J2=     0.000 deg
};
P[30]{
   GP1:
	UF : 1, UT : 1,		CONFIG : 'N U T, 0, 0, 0',
	X =  2103.073  mm,	Y =   282.472  mm,	Z =   462.977  mm,
	W =    30.589 deg,	P =    34.770 deg,	R =    43.796 deg
   GP2:
	UF : 1, UT : 1,
	J1=    90.000 deg,	J2=     0.000 deg
};
P[31]{
   GP1:
	UF : 1, UT : 1,		CONFIG : 'N U T, 0, 0, 0',
	X =  2005.168  mm,	Y =   409.142  mm,	Z =   362.802  mm,
	W =    43.300 deg,	P =    13.762 deg,	R =    75.821 deg
   GP2:
	UF : 1, UT : 1,
	J1=    90.000 deg,	J2=     0.000 deg
};
P[32]{
   GP1:
	UF : 1, UT : 1,		CONFIG : 'N U T, 0, 0, 0',
	X =  2006.405  mm,	Y =   326.766  mm,	Z =   364.251  mm,
	W =    43.298 deg,	P =    13.766 deg,	R =    75.811 deg
   GP2:
	UF : 1, UT : 1,
	J1=    89.999 deg,	J2=     0.000 deg
};
P[33]{
   GP1:
	UF : 1, UT : 1,		CONFIG : 'N U T, 0, 0, 0',
	X =  2084.488  mm,	Y =   314.464  mm,	Z =   441.765  mm,
	W =    43.281 deg,	P =    13.759 deg,	R =    75.826 deg
   GP2:
	UF : 1, UT : 1,
	J1=    90.000 deg,	J2=     0.000 deg
};
P[34]{
   GP1:
	UF : 1, UT : 1,		CONFIG : 'N U T, 0, 0, 0',
	X =  2086.988  mm,	Y =  -331.633  mm,	Z =   441.764  mm,
	W =   -41.228 deg,	P =    19.917 deg,	R =   -68.756 deg
   GP2:
	UF : 1, UT : 1,
	J1=    90.000 deg,	J2=     0.000 deg
};
P[35]{
   GP1:
	UF : 1, UT : 1,		CONFIG : 'N U T, 0, 0, 0',
	X =  2011.652  mm,	Y =  -388.238  mm,	Z =   360.755  mm,
	W =   -41.218 deg,	P =    19.912 deg,	R =   -68.759 deg
   GP2:
	UF : 1, UT : 1,
	J1=    90.000 deg,	J2=     0.000 deg
};
P[36]{
   GP1:
	UF : 1, UT : 1,		CONFIG : 'N U T, 0, 0, 0',
	X =  2009.324  mm,	Y =  -307.165  mm,	Z =   359.779  mm,
	W =   -41.228 deg,	P =    19.919 deg,	R =   -68.761 deg
   GP2:
	UF : 1, UT : 1,
	J1=    90.000 deg,	J2=     0.000 deg
};
P[37]{
   GP1:
	UF : 1, UT : 1,		CONFIG : 'N U T, 0, 0, 0',
	X =  2106.807  mm,	Y =  -322.474  mm,	Z =   465.914  mm,
	W =   -41.228 deg,	P =    19.917 deg,	R =   -68.756 deg
   GP2:
	UF : 1, UT : 1,
	J1=    90.000 deg,	J2=     0.000 deg
};
P[38]{
   GP1:
	UF : 1, UT : 1,		CONFIG : 'N U T, 0, 0, 0',
	X =  2109.307  mm,	Y =    75.081  mm,	Z =   465.913  mm,
	W =     3.207 deg,	P =    44.910 deg,	R =   -85.462 deg
   GP2:
	UF : 1, UT : 1,
	J1=    90.000 deg,	J2=     0.000 deg
};
P[39]{
   GP1:
	UF : 1, UT : 1,		CONFIG : 'N U T, 0, 0, 0',
	X =  2681.306  mm,	Y =  -103.919  mm,	Z =  -438.087  mm,
	W =    -1.257 deg,	P =    33.277 deg,	R =   -88.589 deg
   GP2:
	UF : 1, UT : 1,
	J1=    90.000 deg,	J2=     0.000 deg
};
P[40]{
   GP1:
	UF : 1, UT : 1,		CONFIG : 'N U T, 0, 0, 0',
	X =  2748.326  mm,	Y =   -40.263  mm,	Z =  -588.425  mm,
	W =      .901 deg,	P =    44.837 deg,	R =   -88.538 deg
   GP2:
	UF : 1, UT : 1,
	J1=    89.995 deg,	J2=     0.000 deg
};
P[41]{
   GP1:
	UF : 1, UT : 1,		CONFIG : 'N U T, 0, 0, 0',
	X =  2772.290  mm,	Y =   -39.566  mm,	Z =  -589.780  mm,
	W =      .689 deg,	P =    45.118 deg,	R =   -88.678 deg
   GP2:
	UF : 1, UT : 1,
	J1=    89.993 deg,	J2=     0.000 deg
};
P[42]{
   GP1:
	UF : 1, UT : 1,		CONFIG : 'N U T, 0, 0, 0',
	X =  2676.306  mm,	Y =  -106.919  mm,	Z =  -439.087  mm,
	W =    -1.257 deg,	P =    33.277 deg,	R =   -88.589 deg
   GP2:
	UF : 1, UT : 1,
	J1=    90.000 deg,	J2=     0.000 deg
};
P[43]{
   GP1:
	UF : 1, UT : 1,		CONFIG : 'N U T, 0, 0, 0',
	X =  2576.306  mm,	Y =    -6.919  mm,	Z =  -439.087  mm,
	W =    -1.257 deg,	P =    33.277 deg,	R =   -88.589 deg
   GP2:
	UF : 1, UT : 1,
	J1=    90.000 deg,	J2=     0.000 deg
};
P[44]{
   GP1:
	UF : 1, UT : 1,		CONFIG : 'N U T, 0, 0, 0',
	X =  2582.224  mm,	Y =   118.706  mm,	Z =  -400.809  mm,
	W =      .677 deg,	P =    39.803 deg,	R =    91.170 deg
   GP2:
	UF : 1, UT : 1,
	J1=    90.000 deg,	J2=     0.000 deg
};
P[45]{
   GP1:
	UF : 1, UT : 1,		CONFIG : 'N U T, 0, 0, 0',
	X =  2706.224  mm,	Y =   118.706  mm,	Z =  -483.809  mm,
	W =      .677 deg,	P =    39.803 deg,	R =    91.170 deg
   GP2:
	UF : 1, UT : 1,
	J1=    90.000 deg,	J2=     0.000 deg
};
P[46]{
   GP1:
	UF : 1, UT : 1,		CONFIG : 'N U T, 0, 0, 0',
	X =  2747.106  mm,	Y =    60.104  mm,	Z =  -590.117  mm,
	W =      .903 deg,	P =    44.988 deg,	R =    91.263 deg
   GP2:
	UF : 1, UT : 1,
	J1=    90.000 deg,	J2=     0.000 deg
};
P[47]{
   GP1:
	UF : 1, UT : 1,		CONFIG : 'N U T, 0, 0, 0',
	X =  2767.558  mm,	Y =    60.104  mm,	Z =  -590.117  mm,
	W =      .903 deg,	P =    44.988 deg,	R =    91.263 deg
   GP2:
	UF : 1, UT : 1,
	J1=    90.000 deg,	J2=     0.000 deg
};
P[48]{
   GP1:
	UF : 1, UT : 1,		CONFIG : 'N U T, 0, 0, 0',
	X =  2706.224  mm,	Y =   118.706  mm,	Z =  -483.809  mm,
	W =      .677 deg,	P =    39.803 deg,	R =    91.170 deg
   GP2:
	UF : 1, UT : 1,
	J1=    90.000 deg,	J2=     0.000 deg
};
P[49]{
   GP1:
	UF : 1, UT : 1,		CONFIG : 'N U T, 0, 0, 0',
	X =  2750.938  mm,	Y =   112.285  mm,	Z =  -474.250  mm,
	W =     -.713 deg,	P =    25.922 deg,	R =     -.241 deg
   GP2:
	UF : 1, UT : 1,
	J1=    90.000 deg,	J2=     0.000 deg
};
P[50]{
   GP1:
	UF : 1, UT : 1,		CONFIG : 'N U T, 0, 0, 0',
	X =  2778.081  mm,	Y =    53.285  mm,	Z =  -487.998  mm,
	W =     -.713 deg,	P =    25.922 deg,	R =     -.241 deg
   GP2:
	UF : 1, UT : 1,
	J1=    90.000 deg,	J2=     0.000 deg
};
P[51]{
   GP1:
	UF : 1, UT : 1,		CONFIG : 'N U T, 0, 0, 0',
	X =  2775.833  mm,	Y =    59.955  mm,	Z =  -590.785  mm,
	W =     -.292 deg,	P =    37.605 deg,	R =      .743 deg
   GP2:
	UF : 1, UT : 1,
	J1=    90.000 deg,	J2=     0.000 deg
};
P[52]{
   GP1:
	UF : 1, UT : 1,		CONFIG : 'N U T, 0, 0, 0',
	X =  2775.834  mm,	Y =   -36.401  mm,	Z =  -590.784  mm,
	W =     -.292 deg,	P =    37.605 deg,	R =      .743 deg
   GP2:
	UF : 1, UT : 1,
	J1=    90.000 deg,	J2=     0.000 deg
};
P[53]{
   GP1:
	UF : 1, UT : 1,		CONFIG : 'N U T, 0, 0, 0',
	X =  2774.367  mm,	Y =   -45.046  mm,	Z =  -326.584  mm,
	W =     -.063 deg,	P =     6.406 deg,	R =     -.319 deg
   GP2:
	UF : 1, UT : 1,
	J1=    90.000 deg,	J2=     0.000 deg
};
P[54]{
   GP1:
	UF : 1, UT : 1,		CONFIG : 'N U T, 0, 0, 0',
	X =  2318.510  mm,	Y =     4.126  mm,	Z =   836.416  mm,
	W =     -.063 deg,	P =     6.406 deg,	R =     -.319 deg
   GP2:
	UF : 1, UT : 1,
	J1=    90.000 deg,	J2=     0.000 deg
};
P[55]{
   GP1:
	UF : 1, UT : 1,		CONFIG : 'N U T, 0, 0, 0',
	X =  2651.064  mm,	Y =   274.146  mm,	Z =   596.222  mm,
	W =    40.438 deg,	P =    -1.956 deg,	R =     2.337 deg
   GP2:
	UF : 1, UT : 1,
	J1=    90.000 deg,	J2=     0.000 deg
};
P[56]{
   GP1:
	UF : 1, UT : 1,		CONFIG : 'N U T, 0, 0, 0',
	X =  2678.366  mm,	Y =   323.391  mm,	Z =   552.416  mm,
	W =    40.027 deg,	P =    -6.599 deg,	R =     7.835 deg
   GP2:
	UF : 1, UT : 1,
	J1=    90.000 deg,	J2=     0.000 deg
};
P[57]{
   GP1:
	UF : 1, UT : 1,		CONFIG : 'N U T, 0, 0, 0',
	X =  2749.821  mm,	Y =   428.939  mm,	Z =   464.667  mm,
	W =    44.528 deg,	P =    -7.216 deg,	R =     7.296 deg
   GP2:
	UF : 1, UT : 1,
	J1=    90.000 deg,	J2=     0.000 deg
};
P[58]{
   GP1:
	UF : 1, UT : 1,		CONFIG : 'N U T, 0, 0, 0',
	X =  2715.354  mm,	Y =   428.138  mm,	Z =   464.592  mm,
	W =    44.543 deg,	P =    -7.213 deg,	R =     7.268 deg
   GP2:
	UF : 1, UT : 1,
	J1=    90.000 deg,	J2=     0.000 deg
};
P[59]{
   GP1:
	UF : 1, UT : 1,		CONFIG : 'N U T, 0, 0, 0',
	X =  2698.437  mm,	Y =   269.508  mm,	Z =   599.906  mm,
	W =    44.541 deg,	P =    -7.214 deg,	R =     7.272 deg
   GP2:
	UF : 1, UT : 1,
	J1=    90.000 deg,	J2=     0.000 deg
};
P[60]{
   GP1:
	UF : 1, UT : 1,		CONFIG : 'N U T, 0, 0, 0',
	X =  2703.937  mm,	Y =  -282.492  mm,	Z =   602.906  mm,
	W =   -34.404 deg,	P =     5.822 deg,	R =     8.425 deg
   GP2:
	UF : 1, UT : 1,
	J1=    90.000 deg,	J2=     0.000 deg
};
P[61]{
   GP1:
	UF : 1, UT : 1,		CONFIG : 'N U T, 0, 0, 0',
	X =  2752.117  mm,	Y =  -403.442  mm,	Z =   463.818  mm,
	W =   -44.526 deg,	P =     7.212 deg,	R =     7.276 deg
   GP2:
	UF : 1, UT : 1,
	J1=    90.000 deg,	J2=     0.000 deg
};
P[62]{
   GP1:
	UF : 1, UT : 1,		CONFIG : 'N U T, 0, 0, 0',
	X =  2715.282  mm,	Y =  -404.077  mm,	Z =   462.987  mm,
	W =   -44.523 deg,	P =     7.209 deg,	R =     7.270 deg
   GP2:
	UF : 1, UT : 1,
	J1=    90.000 deg,	J2=     0.000 deg
};
P[63]{
   GP1:
	UF : 1, UT : 1,		CONFIG : 'N U T, 0, 0, 0',
	X =  2699.988  mm,	Y =  -282.600  mm,	Z =   597.231  mm,
	W =   -44.541 deg,	P =     7.214 deg,	R =     7.272 deg
   GP2:
	UF : 1, UT : 1,
	J1=    90.000 deg,	J2=     0.000 deg
};
P[64]{
   GP1:
	UF : 1, UT : 1,		CONFIG : 'F U T, 0, 0, 0',
	X =  2542.011  mm,	Y =    62.997  mm,	Z =   733.500  mm,
	W =      .337 deg,	P =   -50.731 deg,	R =     6.061 deg
   GP2:
	UF : 1, UT : 1,
	J1=    90.000 deg,	J2=     0.000 deg
};
P[65]{
   GP1:
	UF : 1, UT : 1,		CONFIG : 'F U T, 0, 0, 0',
	X =  2864.014  mm,	Y =   282.441  mm,	Z =   502.065  mm,
	W =   -15.171 deg,	P =   -43.175 deg,	R =    33.524 deg
   GP2:
	UF : 1, UT : 1,
	J1=    90.000 deg,	J2=     0.000 deg
};
P[66]{
   GP1:
	UF : 1, UT : 1,		CONFIG : 'F U T, 0, 0, 0',
	X =  2905.759  mm,	Y =   297.489  mm,	Z =   466.526  mm,
	W =   -14.926 deg,	P =   -42.904 deg,	R =    33.356 deg
   GP2:
	UF : 1, UT : 1,
	J1=    90.000 deg,	J2=     0.000 deg
};
P[67]{
   GP1:
	UF : 1, UT : 1,		CONFIG : 'F U T, 0, 0, 0',
	X =  2904.895  mm,	Y =   379.659  mm,	Z =   467.464  mm,
	W =    -8.441 deg,	P =   -43.927 deg,	R =    33.763 deg
   GP2:
	UF : 1, UT : 1,
	J1=    90.000 deg,	J2=     0.000 deg
};
P[68]{
   GP1:
	UF : 1, UT : 1,		CONFIG : 'F U T, 0, 0, 0',
	X =  2904.123  mm,	Y =   411.321  mm,	Z =   468.436  mm,
	W =    -2.983 deg,	P =   -44.252 deg,	R =    40.170 deg
   GP2:
	UF : 1, UT : 1,
	J1=    90.000 deg,	J2=     0.000 deg
};
P[69]{
   GP1:
	UF : 1, UT : 1,		CONFIG : 'F U T, 0, 0, 0',
	X =  2902.073  mm,	Y =   421.602  mm,	Z =   467.948  mm,
	W =    -2.617 deg,	P =   -43.939 deg,	R =    53.826 deg
   GP2:
	UF : 1, UT : 1,
	J1=    90.000 deg,	J2=     0.000 deg
};
P[70]{
   GP1:
	UF : 1, UT : 1,		CONFIG : 'F U T, 0, 0, 0',
	X =  2887.593  mm,	Y =   431.459  mm,	Z =   467.662  mm,
	W =    -2.617 deg,	P =   -43.939 deg,	R =    78.094 deg
   GP2:
	UF : 1, UT : 1,
	J1=    90.000 deg,	J2=     0.000 deg
};
P[71]{
   GP1:
	UF : 1, UT : 1,		CONFIG : 'F U T, 0, 0, 0',
	X =  2878.735  mm,	Y =   431.459  mm,	Z =   467.662  mm,
	W =    -2.617 deg,	P =   -43.939 deg,	R =    78.094 deg
   GP2:
	UF : 1, UT : 1,
	J1=    90.000 deg,	J2=     0.000 deg
};
P[72]{
   GP1:
	UF : 1, UT : 1,		CONFIG : 'F U T, 0, 0, 0',
	X =  2697.000  mm,	Y =   247.797  mm,	Z =   648.652  mm,
	W =    -2.629 deg,	P =   -43.936 deg,	R =    42.269 deg
   GP2:
	UF : 1, UT : 1,
	J1=    90.000 deg,	J2=     0.000 deg
};
P[73]{
   GP1:
	UF : 1, UT : 1,		CONFIG : 'N U T, 0, 0, 0',
	X =   949.898  mm,	Y =    98.916  mm,	Z =  1480.357  mm,
	W =   -25.667 deg,	P =   -34.352 deg,	R =    34.753 deg
   GP2:
	UF : 1, UT : 1,
	J1=     0.000 deg,	J2=   180.000 deg
};
P[74]{
   GP1:
	UF : 1, UT : 1,		CONFIG : 'N U T, 1, 0, 0',
	X =  2528.555  mm,	Y =   -65.615  mm,	Z =   892.718  mm,
	W =   -11.578 deg,	P =   -57.733 deg,	R =     8.895 deg
   GP2:
	UF : 1, UT : 1,
	J1=    90.000 deg,	J2=     0.000 deg
};
P[75]{
   GP1:
	UF : 1, UT : 1,		CONFIG : 'N U T, 0, 0, 0',
	X =  2860.056  mm,	Y =  -309.345  mm,	Z =   520.586  mm,
	W =    14.883 deg,	P =   -42.517 deg,	R =   -27.206 deg
   GP2:
	UF : 1, UT : 1,
	J1=    90.000 deg,	J2=     0.000 deg
};
P[76]{
   GP1:
	UF : 1, UT : 1,		CONFIG : 'N U T, 0, 0, 0',
	X =  2903.526  mm,	Y =  -269.076  mm,	Z =   466.198  mm,
	W =    14.881 deg,	P =   -42.512 deg,	R =   -27.203 deg
   GP2:
	UF : 1, UT : 1,
	J1=    90.000 deg,	J2=     0.000 deg
};
P[77]{
   GP1:
	UF : 1, UT : 1,		CONFIG : 'N U T, 0, 0, 0',
	X =  2902.858  mm,	Y =  -366.735  mm,	Z =   467.050  mm,
	W =     7.402 deg,	P =   -43.864 deg,	R =   -27.796 deg
   GP2:
	UF : 1, UT : 1,
	J1=    90.000 deg,	J2=     0.000 deg
};
P[78]{
   GP1:
	UF : 1, UT : 1,		CONFIG : 'N U T, 0, 0, 0',
	X =  2902.317  mm,	Y =  -381.646  mm,	Z =   467.885  mm,
	W =     7.404 deg,	P =   -43.863 deg,	R =   -33.013 deg
   GP2:
	UF : 1, UT : 1,
	J1=    90.000 deg,	J2=     0.000 deg
};
P[79]{
   GP1:
	UF : 1, UT : 1,		CONFIG : 'N U T, 0, 0, 0',
	X =  2895.908  mm,	Y =  -394.691  mm,	Z =   467.867  mm,
	W =    -1.094 deg,	P =   -44.445 deg,	R =   -50.602 deg
   GP2:
	UF : 1, UT : 1,
	J1=    89.996 deg,	J2=     0.000 deg
};
P[80]{
   GP1:
	UF : 1, UT : 1,		CONFIG : 'N U T, 0, 0, 0',
	X =  2889.336  mm,	Y =  -400.456  mm,	Z =   464.138  mm,
	W =    -1.103 deg,	P =   -44.447 deg,	R =   -71.047 deg
   GP2:
	UF : 1, UT : 1,
	J1=    89.995 deg,	J2=     0.000 deg
};
P[81]{
   GP1:
	UF : 1, UT : 1,		CONFIG : 'N U T, 0, 0, 0',
	X =  2877.924  mm,	Y =  -402.031  mm,	Z =   463.256  mm,
	W =    -1.100 deg,	P =   -44.451 deg,	R =   -71.051 deg
   GP2:
	UF : 1, UT : 1,
	J1=    89.995 deg,	J2=     0.000 deg
};
P[82]{
   GP1:
	UF : 1, UT : 1,		CONFIG : 'N U T, 0, 0, 0',
	X =  2690.549  mm,	Y =  -310.856  mm,	Z =   600.282  mm,
	W =     1.613 deg,	P =   -43.868 deg,	R =   -40.404 deg
   GP2:
	UF : 1, UT : 1,
	J1=    90.000 deg,	J2=     0.000 deg
};
P[83]{
   GP1:
	UF : 1, UT : 1,		CONFIG : 'F U T, 0, 0, 0',
	X =  2542.011  mm,	Y =    62.997  mm,	Z =   733.500  mm,
	W =      .337 deg,	P =   -50.731 deg,	R =     6.061 deg
   GP2:
	UF : 1, UT : 1,
	J1=    90.000 deg,	J2=     0.000 deg
};
P[84]{
   GP1:
	UF : 1, UT : 1,		CONFIG : 'F U T, 0, 0, 0',
	X =  2864.014  mm,	Y =   282.441  mm,	Z =   502.065  mm,
	W =   -15.171 deg,	P =   -43.175 deg,	R =    33.524 deg
   GP2:
	UF : 1, UT : 1,
	J1=    90.000 deg,	J2=     0.000 deg
};
P[85]{
   GP1:
	UF : 1, UT : 1,		CONFIG : 'N U T, 0, 0, 0',
	X =  2172.059  mm,	Y =  -149.810  mm,	Z =  -336.475  mm,
	W =    -4.848 deg,	P =     4.640 deg,	R =    10.727 deg
   GP2:
	UF : 1, UT : 1,
	J1=    45.000 deg,	J2=   182.246 deg
};
P[86]{
   GP1:
	UF : 1, UT : 1,		CONFIG : 'N U T, 0, 0, 0',
	X =  1780.474  mm,	Y =    29.584  mm,	Z =   -67.946  mm,
	W =    -4.424 deg,	P =     7.600 deg,	R =    11.037 deg
   GP2:
	UF : 1, UT : 1,
	J1=    45.000 deg,	J2=   182.246 deg
};
P[87]{
   GP1:
	UF : 1, UT : 1,		CONFIG : 'N U T, 0, 0, 0',
	X =  2177.031  mm,	Y =    47.881  mm,	Z =  -336.554  mm,
	W =    -4.848 deg,	P =     4.640 deg,	R =    15.933 deg
   GP2:
	UF : 1, UT : 1,
	J1=    45.000 deg,	J2=   182.246 deg
};
P[88]{
   GP1:
	UF : 1, UT : 1,		CONFIG : 'N U B, 0, 0, 0',
	X =   355.995  mm,	Y =    -2.072  mm,	Z =  2424.048  mm,
	W =      .014 deg,	P =   -40.003 deg,	R =     -.008 deg
   GP2:
	UF : 1, UT : 1,
	J1=    80.000 deg,	J2=    90.000 deg
};
P[89]{
   GP1:
	UF : 1, UT : 1,		CONFIG : 'N U T, 0, 0, 0',
	X =  2298.943  mm,	Y =    15.028  mm,	Z =   995.580  mm,
	W =   -33.416 deg,	P =    -1.271 deg,	R =    34.407 deg
   GP2:
	UF : 1, UT : 1,
	J1=    89.999 deg,	J2=   -90.000 deg
};
P[90]{
   GP1:
	UF : 1, UT : 1,		CONFIG : 'N U B, 0, 0, 0',
	X =   356.010  mm,	Y =    -2.130  mm,	Z =  2424.082  mm,
	W =      .012 deg,	P =   -40.007 deg,	R =     -.013 deg
   GP2:
	UF : 1, UT : 1,
	J1=    90.000 deg,	J2=   -90.000 deg
};
P[91]{
   GP1:
	UF : 1, UT : 1,		CONFIG : 'F U T, 0, 0, 0',
	X =  2701.500  mm,	Y =   248.797  mm,	Z =   650.852  mm,
	W =    -2.629 deg,	P =   -43.936 deg,	R =    42.269 deg
   GP2:
	UF : 1, UT : 1,
	J1=    90.000 deg,	J2=     0.000 deg
};
P[92]{
   GP1:
	UF : 1, UT : 1,		CONFIG : 'F U T, 0, 0, 0',
	X =  2542.011  mm,	Y =    62.997  mm,	Z =   733.500  mm,
	W =      .337 deg,	P =   -50.731 deg,	R =     6.061 deg
   GP2:
	UF : 1, UT : 1,
	J1=    90.000 deg,	J2=     0.000 deg
};
P[93]{
   GP1:
	UF : 1, UT : 1,		CONFIG : 'F U T, 0, 0, 0',
	X =  2864.014  mm,	Y =   282.441  mm,	Z =   502.065  mm,
	W =   -15.171 deg,	P =   -43.175 deg,	R =    33.524 deg
   GP2:
	UF : 1, UT : 1,
	J1=    90.000 deg,	J2=     0.000 deg
};
P[94]{
   GP1:
	UF : 1, UT : 1,		CONFIG : 'N U B, 0, 0, 0',
	X =   356.016  mm,	Y =    -2.054  mm,	Z =  2424.089  mm,
	W =      .020 deg,	P =   -40.008 deg,	R =     -.011 deg
   GP2:
	UF : 1, UT : 1,
	J1=    80.000 deg,	J2=   -90.000 deg
};
P[95]{
   GP1:
	UF : 1, UT : 1,		CONFIG : 'N U T, 0, 0, 1',
	X =  1917.622  mm,	Y =   283.121  mm,	Z =   189.834  mm,
	W =   -26.631 deg,	P =    72.567 deg,	R =   160.596 deg
   GP2:
	UF : 1, UT : 1,
	J1=    80.000 deg,	J2=   -90.000 deg
};
P[96]{
   GP1:
	UF : 1, UT : 1,		CONFIG : 'N U T, 0, 0, 0',
	X =  2849.615  mm,	Y =  1373.219  mm,	Z =    -7.397  mm,
	W =      .303 deg,	P =     1.056 deg,	R =    25.442 deg
   GP2:
	UF : 1, UT : 1,
	J1=    89.998 deg,	J2=    90.000 deg
};
P[97]{
   GP1:
	UF : 1, UT : 1,		CONFIG : 'N U T, 0, 0, 0',
	X =  1913.400  mm,	Y = -1217.274  mm,	Z =  1258.765  mm,
	W =   -40.515 deg,	P =     2.084 deg,	R =   -24.296 deg
   GP2:
	UF : 1, UT : 1,
	J1=   180.000 deg,	J2=   -90.000 deg
};
P[98]{
   GP1:
	UF : 1, UT : 1,		CONFIG : 'N U B, 0, 0, 0',
	X =   355.994  mm,	Y =    -2.149  mm,	Z =  2424.037  mm,
	W =     -.001 deg,	P =   -40.002 deg,	R =     -.003 deg
   GP2:
	UF : 1, UT : 1,
	J1=   180.000 deg,	J2=   -90.000 deg
};
P[99]{
   GP1:
	UF : 1, UT : 1,		CONFIG : 'N U T, 0, 0, 0',
	X =  1419.375  mm,	Y =   870.775  mm,	Z =  1903.281  mm,
	W =    32.261 deg,	P =   -18.474 deg,	R =    10.214 deg
   GP2:
	UF : 1, UT : 1,
	J1=   180.000 deg,	J2=    90.000 deg
};
P[100]{
   GP1:
	UF : 1, UT : 1,		CONFIG : 'F U T, 0, 0, 0',
	X =  2701.500  mm,	Y =   248.797  mm,	Z =   650.852  mm,
	W =    -2.629 deg,	P =   -43.936 deg,	R =    42.269 deg
   GP2:
	UF : 1, UT : 1,
	J1=    90.000 deg,	J2=     0.000 deg
};
P[101]{
   GP1:
	UF : 1, UT : 1,		CONFIG : 'N U T, 0, 0, 0',
	X =  2849.614  mm,	Y =  1359.434  mm,	Z =    -7.398  mm,
	W =      .171 deg,	P =     1.085 deg,	R =    18.410 deg
   GP2:
	UF : 1, UT : 1,
	J1=    89.998 deg,	J2=    90.000 deg
};
P[102]{
   GP1:
	UF : 1, UT : 1,		CONFIG : 'N U T, 0, 0, 0',
	X =  2687.056  mm,	Y =  -231.345  mm,	Z =   639.889  mm,
	W =    14.883 deg,	P =   -42.517 deg,	R =   -27.206 deg
   GP2:
	UF : 1, UT : 1,
	J1=    90.000 deg,	J2=     0.000 deg
};
P[103]{
   GP1:
	UF : 1, UT : 1,		CONFIG : 'N U T, 0, 0, 0',
	X =  2860.056  mm,	Y =  -309.345  mm,	Z =   520.586  mm,
	W =    14.883 deg,	P =   -42.517 deg,	R =   -27.206 deg
   GP2:
	UF : 1, UT : 1,
	J1=    90.000 deg,	J2=     0.000 deg
};
P[104]{
   GP1:
	UF : 1, UT : 1,		CONFIG : 'N U B, 0, 0, 0',
	X =   356.007  mm,	Y =    -2.068  mm,	Z =  2424.055  mm,
	W =      .010 deg,	P =   -40.003 deg,	R =     -.004 deg
   GP2:
	UF : 1, UT : 1,
	J1=   180.000 deg,	J2=   150.000 deg
};
P[105]{
   GP1:
	UF : 1, UT : 1,		CONFIG : 'N U T, 0, 0, 0',
	X =  1166.553  mm,	Y = -1374.013  mm,	Z =  1522.225  mm,
	W =   -32.586 deg,	P =   -12.067 deg,	R =    17.529 deg
   GP2:
	UF : 1, UT : 1,
	J1=   180.000 deg,	J2=  -125.000 deg
};
P[106]{
   GP1:
	UF : 1, UT : 1,		CONFIG : 'N U T, 0, 0, 0',
	X =  2337.765  mm,	Y = -1447.908  mm,	Z =  1189.179  mm,
	W =   -45.668 deg,	P =   -29.178 deg,	R =    61.340 deg
   GP2:
	UF : 1, UT : 1,
	J1=   100.000 deg,	J2=   -90.000 deg
};
P[107]{
   GP1:
	UF : 1, UT : 1,		CONFIG : 'N U B, 0, 0, 0',
	X =   347.064  mm,	Y =    -5.448  mm,	Z =  2436.079  mm,
	W =     -.019 deg,	P =   -39.997 deg,	R =      .013 deg
   GP2:
	UF : 1, UT : 1,
	J1=   100.000 deg,	J2=   -90.000 deg
};
P[108]{
   GP1:
	UF : 1, UT : 1,		CONFIG : 'N U T, 0, 0, 0',
	X =  1642.115  mm,	Y = -1225.593  mm,	Z =  1744.283  mm,
	W =   -30.785 deg,	P =   -19.925 deg,	R =    38.701 deg
   GP2:
	UF : 1, UT : 1,
	J1=   100.000 deg,	J2=   -90.000 deg
};
P[109]{
   GP1:
	UF : 1, UT : 1,		CONFIG : 'N U T, 0, 0, 0',
	X =  2337.765  mm,	Y = -1447.908  mm,	Z =  1189.179  mm,
	W =   -45.668 deg,	P =   -29.178 deg,	R =    61.340 deg
   GP2:
	UF : 1, UT : 1,
	J1=   100.000 deg,	J2=   -90.000 deg
};
P[110]{
   GP1:
	UF : 1, UT : 1,		CONFIG : 'N U T, 0, 0, 0',
	X =  2690.549  mm,	Y =  -310.856  mm,	Z =   600.282  mm,
	W =     1.613 deg,	P =   -43.868 deg,	R =   -40.404 deg
   GP2:
	UF : 1, UT : 1,
	J1=    90.000 deg,	J2=     0.000 deg
};
P[111]{
   GP1:
	UF : 1, UT : 1,		CONFIG : 'N U T, 1, 0, 0',
	X =  2528.555  mm,	Y =   -65.615  mm,	Z =   892.718  mm,
	W =   -11.578 deg,	P =   -57.733 deg,	R =     8.895 deg
   GP2:
	UF : 1, UT : 1,
	J1=    90.000 deg,	J2=     0.000 deg
};
P[112]{
   GP1:
	UF : 1, UT : 1,		CONFIG : 'N U T, 0, 0, 0',
	X =  2860.056  mm,	Y =  -309.345  mm,	Z =   520.586  mm,
	W =    14.883 deg,	P =   -42.517 deg,	R =   -27.206 deg
   GP2:
	UF : 1, UT : 1,
	J1=    90.000 deg,	J2=     0.000 deg
};
P[113]{
   GP1:
	UF : 1, UT : 1,		CONFIG : 'N U T, 0, 0, 0',
	X =  1539.625  mm,	Y = -1470.562  mm,	Z =  1075.975  mm,
	W =   -42.854 deg,	P =   -15.295 deg,	R =    39.123 deg
   GP2:
	UF : 1, UT : 1,
	J1=   180.000 deg,	J2=  -125.000 deg
};
P[114]{
   GP1:
	UF : 1, UT : 1,		CONFIG : 'N U B, 0, 0, 0',
	X =   356.032  mm,	Y =    -2.146  mm,	Z =  2424.049  mm,
	W =      .001 deg,	P =   -40.002 deg,	R =     -.005 deg
   GP2:
	UF : 1, UT : 1,
	J1=    95.000 deg,	J2=    90.000 deg
};
P[115]{
   GP1:
	UF : 1, UT : 1,		CONFIG : 'N U T, 0, 0, 0',
	X =  2048.592  mm,	Y =  1142.742  mm,	Z =  1844.585  mm,
	W =    41.764 deg,	P =     3.536 deg,	R =   -26.914 deg
   GP2:
	UF : 1, UT : 1,
	J1=    95.000 deg,	J2=    90.000 deg
};
P[116]{
   GP1:
	UF : 1, UT : 1,		CONFIG : 'N U B, 0, 0, 0',
	X =   356.004  mm,	Y =    -2.058  mm,	Z =  2424.066  mm,
	W =      .021 deg,	P =   -40.005 deg,	R =     -.012 deg
   GP2:
	UF : 1, UT : 1,
	J1=   125.000 deg,	J2=     0.000 deg
};
P[117]{
   GP1:
	UF : 1, UT : 1,		CONFIG : 'N U B, 0, 0, 0',
	X =   356.032  mm,	Y =    -2.146  mm,	Z =  2424.050  mm,
	W =      .001 deg,	P =   -40.002 deg,	R =     -.005 deg
   GP2:
	UF : 1, UT : 1,
	J1=     0.000 deg,	J2=   180.000 deg
};
P[118]{
   GP1:
	UF : 1, UT : 1,		CONFIG : 'N U B, 0, 0, 0',
	X =   356.032  mm,	Y =    -2.146  mm,	Z =  2424.049  mm,
	W =      .001 deg,	P =   -40.002 deg,	R =     -.005 deg
   GP2:
	UF : 1, UT : 1,
	J1=    90.000 deg,	J2=    90.000 deg
};
P[119]{
   GP1:
	UF : 1, UT : 1,		CONFIG : 'N U T, 0, 0, 0',
	X =  2690.549  mm,	Y =  -310.856  mm,	Z =   600.282  mm,
	W =     1.613 deg,	P =   -43.868 deg,	R =   -40.404 deg
   GP2:
	UF : 1, UT : 1,
	J1=    90.000 deg,	J2=     0.000 deg
};
P[120]{
   GP1:
	UF : 1, UT : 1,		CONFIG : 'N U T, 0, 0, 0',
	X =  2831.471  mm,	Y =  1359.434  mm,	Z =    -7.398  mm,
	W =      .171 deg,	P =     1.085 deg,	R =    18.410 deg
   GP2:
	UF : 1, UT : 1,
	J1=    89.998 deg,	J2=    90.000 deg
};
P[121]{
   GP1:
	UF : 1, UT : 1,		CONFIG : 'N U T, 0, 0, -1',
	X =  2671.361  mm,	Y =  -220.509  mm,	Z =   618.788  mm,
	W =    39.952 deg,	P =    49.905 deg,	R =  -159.452 deg
   GP2:
	UF : 1, UT : 1,
	J1=    90.000 deg,	J2=     0.000 deg
};
P[122]{
   GP1:
	UF : 1, UT : 1,		CONFIG : 'N U T, 0, 0, 0',
	X =  2675.436  mm,	Y =  -298.605  mm,	Z =   591.354  mm,
	W =    31.909 deg,	P =    33.590 deg,	R =  -130.034 deg
   GP2:
	UF : 1, UT : 1,
	J1=    90.000 deg,	J2=     0.000 deg
};
P[123]{
   GP1:
	UF : 1, UT : 1,		CONFIG : 'N U T, 0, 0, 0',
	X =  2831.470  mm,	Y =  1380.434  mm,	Z =    -7.398  mm,
	W =      .171 deg,	P =     1.085 deg,	R =    18.410 deg
   GP2:
	UF : 1, UT : 1,
	J1=    89.998 deg,	J2=    90.000 deg
};
P[124]{
   GP1:
	UF : 1, UT : 1,		CONFIG : 'N U T, 0, 0, 0',
	X =  1269.879  mm,	Y = -1253.433  mm,	Z =    79.373  mm,
	W =    -1.683 deg,	P =    44.139 deg,	R =  -145.609 deg
   GP2:
	UF : 1, UT : 1,
	J1=     0.000 deg,	J2=   -40.000 deg
};
P[125]{
   GP1:
	UF : 1, UT : 1,		CONFIG : 'N U T, 0, 0, 0',
	X =  1314.620  mm,	Y = -1313.270  mm,	Z =    82.919  mm,
	W =     1.498 deg,	P =    44.726 deg,	R =  -177.480 deg
   GP2:
	UF : 1, UT : 1,
	J1=     0.000 deg,	J2=   -40.000 deg
};
P[126]{
   GP1:
	UF : 1, UT : 1,		CONFIG : 'N U T, 0, 0, 0',
	X =   907.923  mm,	Y =  -828.465  mm,	Z =    78.992  mm,
	W =     -.234 deg,	P =    44.187 deg,	R =  -138.544 deg
   GP2:
	UF : 1, UT : 1,
	J1=     0.000 deg,	J2=   -40.000 deg
};
P[127]{
   GP1:
	UF : 1, UT : 1,		CONFIG : 'N U T, 0, 0, 0',
	X =  2781.851  mm,	Y =  -350.503  mm,	Z =   533.590  mm,
	W =    31.150 deg,	P =     5.212 deg,	R =   -83.519 deg
   GP2:
	UF : 1, UT : 1,
	J1=    90.000 deg,	J2=     0.000 deg
};
P[128]{
   GP1:
	UF : 1, UT : 1,		CONFIG : 'N U T, 0, 0, 0',
	X =  2698.335  mm,	Y =   256.194  mm,	Z =   573.763  mm,
	W =   -42.051 deg,	P =    32.739 deg,	R =   124.663 deg
   GP2:
	UF : 1, UT : 1,
	J1=    90.000 deg,	J2=     0.000 deg
};
P[129]{
   GP1:
	UF : 1, UT : 1,		CONFIG : 'N U T, 0, 0, 0',
	X =  1239.992  mm,	Y = -1224.689  mm,	Z =    81.310  mm,
	W =      .993 deg,	P =    44.648 deg,	R =  -147.123 deg
   GP2:
	UF : 1, UT : 1,
	J1=     0.000 deg,	J2=   -40.000 deg
};
P[130]{
   GP1:
	UF : 1, UT : 1,		CONFIG : 'N U T, 0, 0, 0',
	X =   882.027  mm,	Y =  -793.098  mm,	Z =    83.021  mm,
	W =    -1.714 deg,	P =    41.650 deg,	R =  -137.126 deg
   GP2:
	UF : 1, UT : 1,
	J1=     0.000 deg,	J2=   -40.000 deg
};
P[131]{
   GP1:
	UF : 1, UT : 1,		CONFIG : 'N U T, 0, 0, 0',
	X =   833.656  mm,	Y =  -734.388  mm,	Z =    84.663  mm,
	W =    -1.870 deg,	P =    41.238 deg,	R =  -117.739 deg
   GP2:
	UF : 1, UT : 1,
	J1=     0.000 deg,	J2=   -40.000 deg
};
P[132]{
   GP1:
	UF : 1, UT : 1,		CONFIG : 'N U T, 0, 0, 0',
	X =  2507.432  mm,	Y =   427.190  mm,	Z =   497.403  mm,
	W =    44.780 deg,	P =     5.017 deg,	R =    -1.188 deg
   GP2:
	UF : 1, UT : 1,
	J1=    90.000 deg,	J2=     0.000 deg
};
P[133]{
   GP1:
	UF : 1, UT : 1,		CONFIG : 'N U T, 0, 0, 0',
	X =  2750.496  mm,	Y =   369.295  mm,	Z =   531.685  mm,
	W =   -32.204 deg,	P =    27.169 deg,	R =   115.020 deg
   GP2:
	UF : 1, UT : 1,
	J1=    90.000 deg,	J2=     0.000 deg
};
P[134]{
   GP1:
	UF : 1, UT : 1,		CONFIG : 'N U T, 0, 0, 0',
	X =  2433.364  mm,	Y =   -19.547  mm,	Z =   530.114  mm,
	W =    -7.526 deg,	P =    51.572 deg,	R =   125.549 deg
   GP2:
	UF : 1, UT : 1,
	J1=    90.000 deg,	J2=     0.000 deg
};
P[135]{
   GP1:
	UF : 1, UT : 1,		CONFIG : 'N U T, 0, 0, 0',
	X =  1964.092  mm,	Y =   128.072  mm,	Z =   485.282  mm,
	W =    14.025 deg,	P =    31.485 deg,	R =    29.572 deg
   GP2:
	UF : 1, UT : 1,
	J1=    90.000 deg,	J2=     0.000 deg
};
P[136]{
   GP1:
	UF : 1, UT : 1,		CONFIG : 'N U T, 0, 0, 0',
	X =  1776.950  mm,	Y =   181.788  mm,	Z =   449.993  mm,
	W =    35.022 deg,	P =    36.482 deg,	R =    50.220 deg
   GP2:
	UF : 1, UT : 1,
	J1=    90.000 deg,	J2=     0.000 deg
};
P[137]{
   GP1:
	UF : 1, UT : 1,		CONFIG : 'N U T, 0, 0, 0',
	X =  2456.052  mm,	Y =   425.683  mm,	Z =   498.220  mm,
	W =    45.076 deg,	P =     5.046 deg,	R =    -1.313 deg
   GP2:
	UF : 1, UT : 1,
	J1=    89.999 deg,	J2=     0.000 deg
};
P[138]{
   GP1:
	UF : 1, UT : 1,		CONFIG : 'N U T, 0, 0, 0',
	X =  2440.584  mm,	Y =   427.227  mm,	Z =   496.365  mm,
	W =    44.794 deg,	P =     5.016 deg,	R =    30.070 deg
   GP2:
	UF : 1, UT : 1,
	J1=    90.000 deg,	J2=     0.000 deg
};
P[139]{
   GP1:
	UF : 1, UT : 1,		CONFIG : 'N U T, 0, 0, 0',
	X =  1754.079  mm,	Y =   165.415  mm,	Z =   449.266  mm,
	W =    31.721 deg,	P =    33.769 deg,	R =    48.036 deg
   GP2:
	UF : 1, UT : 1,
	J1=    90.000 deg,	J2=     0.000 deg
};
P[140]{
   GP1:
	UF : 1, UT : 1,		CONFIG : 'N U T, 0, 0, 0',
	X =  1754.079  mm,	Y =  -235.814  mm,	Z =   449.266  mm,
	W =   -34.074 deg,	P =    31.387 deg,	R =   -52.404 deg
   GP2:
	UF : 1, UT : 1,
	J1=    90.000 deg,	J2=     0.000 deg
};
P[141]{
   GP1:
	UF : 1, UT : 1,		CONFIG : 'N U T, 0, 0, 0',
	X =  2524.023  mm,	Y =  -405.057  mm,	Z =   494.826  mm,
	W =   -44.056 deg,	P =    10.309 deg,	R =     9.167 deg
   GP2:
	UF : 1, UT : 1,
	J1=    90.000 deg,	J2=     0.000 deg
};
P[142]{
   GP1:
	UF : 1, UT : 1,		CONFIG : 'N U T, 0, 0, 0',
	X =  2485.759  mm,	Y =  -405.522  mm,	Z =   494.261  mm,
	W =   -44.059 deg,	P =    10.320 deg,	R =     9.160 deg
   GP2:
	UF : 1, UT : 1,
	J1=    90.000 deg,	J2=     0.000 deg
};
P[143]{
   GP1:
	UF : 1, UT : 1,		CONFIG : 'N U T, 0, 0, 0',
	X =  1843.198  mm,	Y =  -173.825  mm,	Z =   537.934  mm,
	W =   -34.074 deg,	P =    31.387 deg,	R =   -52.404 deg
   GP2:
	UF : 1, UT : 1,
	J1=    90.000 deg,	J2=     0.000 deg
};
P[144]{
   GP1:
	UF : 1, UT : 1,		CONFIG : 'N U T, 0, 0, 0',
	X =  1807.054  mm,	Y =   -90.826  mm,	Z =  1125.220  mm,
	W =      .036 deg,	P =     1.106 deg,	R =     1.891 deg
   GP2:
	UF : 1, UT : 1,
	J1=    45.000 deg,	J2=     0.000 deg
};
P[145]{
   GP1:
	UF : 1, UT : 1,		CONFIG : 'N U T, 0, 0, 0',
	X =  1807.054  mm,	Y =  -390.825  mm,	Z =  1004.220  mm,
	W =     -.607 deg,	P =      .924 deg,	R =   -33.344 deg
   GP2:
	UF : 1, UT : 1,
	J1=    45.000 deg,	J2=     0.000 deg
};
P[146]{
   GP1:
	UF : 1, UT : 1,		CONFIG : 'N U T, 0, 0, 0',
	X =  2449.237  mm,	Y =  -403.696  mm,	Z =   493.863  mm,
	W =   -44.053 deg,	P =    10.305 deg,	R =   -21.685 deg
   GP2:
	UF : 1, UT : 1,
	J1=    90.000 deg,	J2=     0.000 deg
};
P[147]{
   GP1:
	UF : 1, UT : 1,		CONFIG : 'N U T, 0, 0, 0',
	X =  2005.168  mm,	Y =   409.142  mm,	Z =   362.802  mm,
	W =    43.300 deg,	P =    13.762 deg,	R =    75.821 deg
   GP2:
	UF : 1, UT : 1,
	J1=    90.000 deg,	J2=     0.000 deg
};
P[148]{
   GP1:
	UF : 1, UT : 1,		CONFIG : 'N U T, 0, 0, 0',
	X =  1816.054  mm,	Y =  -176.826  mm,	Z =  1084.220  mm,
	W =     -.607 deg,	P =      .924 deg,	R =   -33.344 deg
   GP2:
	UF : 1, UT : 1,
	J1=    45.000 deg,	J2=     0.000 deg
};
P[149]{
   GP1:
	UF : 1, UT : 1,		CONFIG : 'N U T, 0, 0, 0',
	X =  1807.054  mm,	Y =   376.174  mm,	Z =  1018.220  mm,
	W =     -.607 deg,	P =      .924 deg,	R =    40.441 deg
   GP2:
	UF : 1, UT : 1,
	J1=    45.000 deg,	J2=     0.000 deg
};
P[150]{
   GP1:
	UF : 1, UT : 1,		CONFIG : 'N U T, 0, 0, 0',
	X =  2006.405  mm,	Y =   326.766  mm,	Z =   364.251  mm,
	W =    43.298 deg,	P =    13.766 deg,	R =    75.811 deg
   GP2:
	UF : 1, UT : 1,
	J1=    89.999 deg,	J2=     0.000 deg
};
P[151]{
   GP1:
	UF : 1, UT : 1,		CONFIG : 'N U T, 0, 0, 0',
	X =  2011.652  mm,	Y =  -388.238  mm,	Z =   360.755  mm,
	W =   -41.218 deg,	P =    19.912 deg,	R =   -68.759 deg
   GP2:
	UF : 1, UT : 1,
	J1=    90.000 deg,	J2=     0.000 deg
};
P[152]{
   GP1:
	UF : 1, UT : 1,		CONFIG : 'N U T, 0, 0, 0',
	X =  1807.054  mm,	Y =   173.895  mm,	Z =  1166.219  mm,
	W =     -.607 deg,	P =      .924 deg,	R =    40.441 deg
   GP2:
	UF : 1, UT : 1,
	J1=    45.000 deg,	J2=     0.000 deg
};
P[153]{
   GP1:
	UF : 1, UT : 1,		CONFIG : 'N U T, 0, 0, 0',
	X =   908.243  mm,	Y =     -.972  mm,	Z =  2177.323  mm,
	W =     -.010 deg,	P =   -45.000 deg,	R =     0.000 deg
   GP2:
	UF : 1, UT : 1,
	J1=   125.000 deg,	J2=     0.000 deg
};
P[154]{
   GP1:
	UF : 1, UT : 1,		CONFIG : 'N U T, 0, 0, 0',
	X =  1841.244  mm,	Y =   574.028  mm,	Z =  1589.322  mm,
	W =     -.010 deg,	P =   -11.091 deg,	R =     0.000 deg
   GP2:
	UF : 1, UT : 1,
	J1=   125.000 deg,	J2=     0.000 deg
};
P[155]{
   GP1:
	UF : 1, UT : 1,		CONFIG : 'N U T, 0, 0, 0',
	X =  2130.244  mm,	Y =   574.028  mm,	Z =  1472.322  mm,
	W =     -.010 deg,	P =   -11.091 deg,	R =     0.000 deg
   GP2:
	UF : 1, UT : 1,
	J1=   125.000 deg,	J2=     0.000 deg
};
P[156]{
   GP1:
	UF : 1, UT : 1,		CONFIG : 'N U T, 0, 0, 0',
	X =  2009.324  mm,	Y =  -307.165  mm,	Z =   359.779  mm,
	W =   -41.228 deg,	P =    19.919 deg,	R =   -68.761 deg
   GP2:
	UF : 1, UT : 1,
	J1=    90.000 deg,	J2=     0.000 deg
};
P[157]{
   GP1:
	UF : 1, UT : 1,		CONFIG : 'N U T, 0, 0, 0',
	X =  2748.326  mm,	Y =   -40.263  mm,	Z =  -588.425  mm,
	W =      .901 deg,	P =    44.837 deg,	R =   -88.538 deg
   GP2:
	UF : 1, UT : 1,
	J1=    89.995 deg,	J2=     0.000 deg
};
P[158]{
   GP1:
	UF : 1, UT : 1,		CONFIG : 'N U T, 0, 0, 0',
	X =  2772.290  mm,	Y =   -39.566  mm,	Z =  -589.780  mm,
	W =      .689 deg,	P =    45.118 deg,	R =   -88.678 deg
   GP2:
	UF : 1, UT : 1,
	J1=    89.993 deg,	J2=     0.000 deg
};
P[159]{
   GP1:
	UF : 1, UT : 1,		CONFIG : 'N U T, 0, 0, 0',
	X =  2192.055  mm,	Y =   448.511  mm,	Z =  1378.272  mm,
	W =     0.000 deg,	P =    -1.567 deg,	R =     0.000 deg
   GP2:
	UF : 1, UT : 1,
	J1=   125.000 deg,	J2=     0.000 deg
};
P[160]{
   GP1:
	UF : 1, UT : 1,		CONFIG : 'N U T, 0, 0, 0',
	X =  2174.054  mm,	Y =    17.763  mm,	Z =  1379.272  mm,
	W =     0.000 deg,	P =    -1.567 deg,	R =     0.000 deg
   GP2:
	UF : 1, UT : 1,
	J1=   125.000 deg,	J2=     0.000 deg
};
P[161]{
   GP1:
	UF : 1, UT : 1,		CONFIG : 'N U T, 0, 0, 0',
	X =  2747.106  mm,	Y =    60.104  mm,	Z =  -590.117  mm,
	W =      .903 deg,	P =    44.988 deg,	R =    91.263 deg
   GP2:
	UF : 1, UT : 1,
	J1=    90.000 deg,	J2=     0.000 deg
};
P[162]{
   GP1:
	UF : 1, UT : 1,		CONFIG : 'N U T, 0, 0, 0',
	X =  2767.558  mm,	Y =    60.104  mm,	Z =  -590.117  mm,
	W =      .903 deg,	P =    44.988 deg,	R =    91.263 deg
   GP2:
	UF : 1, UT : 1,
	J1=    90.000 deg,	J2=     0.000 deg
};
P[163]{
   GP1:
	UF : 1, UT : 1,		CONFIG : 'N U T, 0, 0, 0',
	X =  2194.122  mm,	Y =  -401.237  mm,	Z =  1396.402  mm,
	W =     0.000 deg,	P =     1.835 deg,	R =     0.000 deg
   GP2:
	UF : 1, UT : 1,
	J1=   125.000 deg,	J2=     0.000 deg
};
P[164]{
   GP1:
	UF : 1, UT : 1,		CONFIG : 'N U T, 0, 0, 0',
	X =  2176.122  mm,	Y =   354.763  mm,	Z =  1397.402  mm,
	W =     0.000 deg,	P =     1.835 deg,	R =     0.000 deg
   GP2:
	UF : 1, UT : 1,
	J1=   125.000 deg,	J2=     0.000 deg
};
P[165]{
   GP1:
	UF : 1, UT : 1,		CONFIG : 'N U T, 0, 0, 1',
	X =  2745.545  mm,	Y =  -276.052  mm,	Z =   464.654  mm,
	W =    29.147 deg,	P =    30.453 deg,	R =  -132.266 deg
   GP2:
	UF : 1, UT : 1,
	J1=    90.000 deg,	J2=     0.000 deg
};
P[166]{
   GP1:
	UF : 1, UT : 1,		CONFIG : 'N U T, 0, 0, 1',
	X =  2745.001  mm,	Y =  -318.060  mm,	Z =   465.700  mm,
	W =    29.459 deg,	P =    30.698 deg,	R =  -132.107 deg
   GP2:
	UF : 1, UT : 1,
	J1=    90.000 deg,	J2=     0.000 deg
};
P[167]{
   GP1:
	UF : 1, UT : 1,		CONFIG : 'N U T, 0, 0, 0',
	X =  2176.122  mm,	Y =    15.763  mm,	Z =  1427.402  mm,
	W =     0.000 deg,	P =    -4.591 deg,	R =     0.000 deg
   GP2:
	UF : 1, UT : 1,
	J1=   125.000 deg,	J2=     0.000 deg
};
P[168]{
   GP1:
	UF : 1, UT : 1,		CONFIG : 'N U T, 0, 0, 0',
	X =  2176.122  mm,	Y =  -553.165  mm,	Z =  1427.402  mm,
	W =     0.000 deg,	P =    -4.591 deg,	R =     0.000 deg
   GP2:
	UF : 1, UT : 1,
	J1=   125.000 deg,	J2=     0.000 deg
};
P[169]{
   GP1:
	UF : 1, UT : 1,		CONFIG : 'N U T, 0, 0, 1',
	X =  2759.258  mm,	Y =  -343.755  mm,	Z =   464.873  mm,
	W =    32.708 deg,	P =    26.756 deg,	R =  -103.211 deg
   GP2:
	UF : 1, UT : 1,
	J1=    90.000 deg,	J2=     0.000 deg
};
P[170]{
   GP1:
	UF : 1, UT : 1,		CONFIG : 'N U T, 0, 0, 0',
	X =  2781.851  mm,	Y =  -350.503  mm,	Z =   466.805  mm,
	W =    32.871 deg,	P =    19.630 deg,	R =   -83.146 deg
   GP2:
	UF : 1, UT : 1,
	J1=    90.000 deg,	J2=     0.000 deg
};
P[171]{
   GP1:
	UF : 1, UT : 1,		CONFIG : 'N U T, 0, 0, 0',
	X =  2740.523  mm,	Y =   300.010  mm,	Z =   465.528  mm,
	W =   -36.614 deg,	P =    28.247 deg,	R =   122.490 deg
   GP2:
	UF : 1, UT : 1,
	J1=    90.000 deg,	J2=     0.000 deg
};
P[172]{
   GP1:
	UF : 1, UT : 1,		CONFIG : 'N U T, 0, 0, 0',
	X =  2174.639  mm,	Y =  -639.399  mm,	Z =  1514.172  mm,
	W =     0.000 deg,	P =   -23.113 deg,	R =     0.000 deg
   GP2:
	UF : 1, UT : 1,
	J1=   125.000 deg,	J2=     0.000 deg
};
P[173]{
   GP1:
	UF : 1, UT : 1,		CONFIG : 'N U T, 0, 0, 0',
	X =  1929.795  mm,	Y =  -639.399  mm,	Z =  1514.172  mm,
	W =     0.000 deg,	P =   -23.113 deg,	R =     0.000 deg
   GP2:
	UF : 1, UT : 1,
	J1=   125.000 deg,	J2=     0.000 deg
};
P[174]{
   GP1:
	UF : 1, UT : 1,		CONFIG : 'N U B, 0, 0, 0',
	X =   356.032  mm,	Y =    -2.146  mm,	Z =  2424.050  mm,
